RoboDK station: kr30 cnc 070419 2.rdk

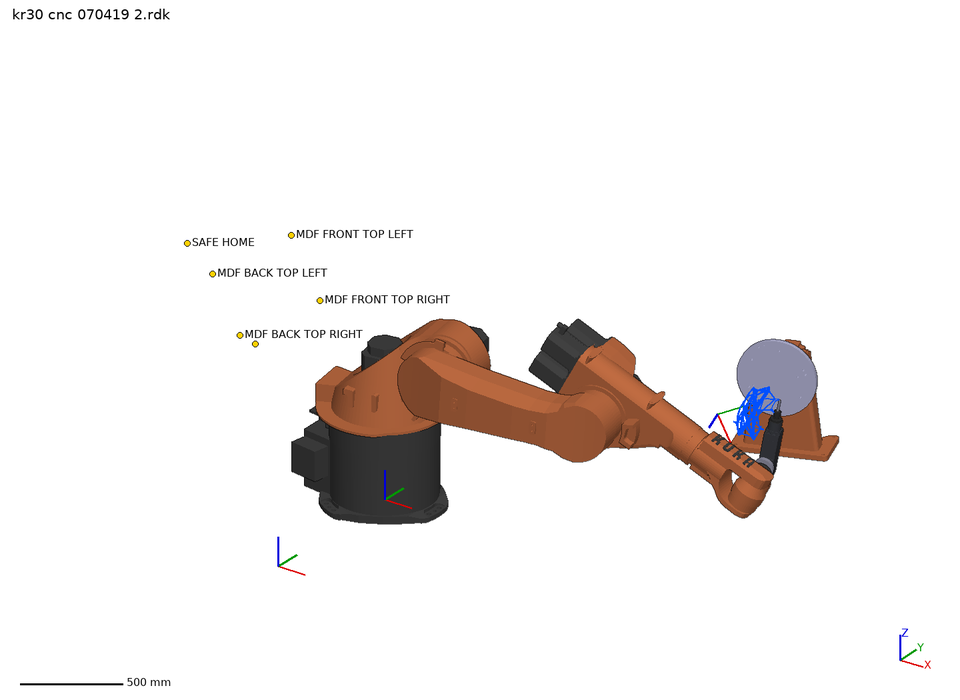
[picture v0: the station drawn from its stored meshes, robots at their saved joint values, targets as dots, program paths as lines]
Station kr30 cnc 070419 2. Poses are relative to the parent item; angles as X-Y-Z fixed-axis rotations.
  - frame GIGASHEEN 7th Axis Base at (0, 1100, 0) mm
    - robot KUKA KP1 MD250: 1 axes, payload 250 kg
        modified DH rows (alpha deg, a mm, theta deg, d mm): 0, 0, 0, 0
        base shift (1750, 1710, 820) mm, rotated rx 0 ry 90 rz -70 deg
        joint limits [-3600] to [3600]; home [0]; saved at [-335.665]
      - frame Reference Rhino at (0, -250, 250) mm
        - object RhinoPart at (0, 0, 0) mm
  - frame GIGASHEEN Base at (0, 2000, 0) mm
    - robot GIGASHEEN (model KUKA KR 30 HA): 6 axes, payload 30 kg, reach 2033 mm, repeatability 0.05 mm, weight 665 kg
        modified DH rows (alpha deg, a mm, theta deg, d mm): 0, 0, 0, 815; -90, 350, 0, 0; 0, 850, -90, 0; -90, 145, 0, 820; 90, 0, 0, 0; -90, 0, 180, 170
        joint limits [-185, -135, -120, -350, -119, -350] to [185, 35, 158, 350, 119, 350]; home [0, -90, 90, 0, 0, 0]; saved at [-7.883, 4.087, 23.625, 95.701, -100.709, 108.247]
      - tool 1/2" End Mill TCP, TCP at (337.71, -2.2, 160.57) mm, rotated rx 0 ry 90 rz 0 deg, size 415.8 x 102 x 153.6 mm
    - target MDF BACK TOP LEFT (joint target) at (-335.18, -974.02, 1512.92) mm, rotated rx 85.17 ry 71.84 rz 47.05 deg; joints [27.716, -45.008, 102.25, 116.233, 75.695, -151.59, -681.46] of GIGASHEEN
    - target MDF FRONT TOP LEFT (joint target) at (-87.97, -665.25, 1668.52) mm, rotated rx 85.17 ry 71.84 rz 47.05 deg; joints [22.06, -21.631, 54.581, 104.768, 70.881, -126.376, -681.46] of GIGASHEEN
    - target MDF FRONT TOP RIGHT (joint target) at (4.03, -550.6, 1295.2) mm, rotated rx 85.17 ry 71.84 rz 47.05 deg; joints [10.053, -29.315, 70.245, 98.928, 81.917, -132.341, -681.46] of GIGASHEEN
    - target MDF BACK TOP RIGHT (joint target) at (-248.73, -867.72, 1165.36) mm, rotated rx 85.17 ry 71.84 rz 47.05 deg; joints [13.787, -50.344, 113.459, 104.66, 84.215, -154.683, -681.46] of GIGASHEEN
    - target MDF STOCK DEPTH (only use z axis value) (joint target) at (-166.67, -856.91, 1136.76) mm, rotated rx 85.17 ry 71.84 rz 47.05 deg; joints [11.502, -45.737, 110.222, 102.707, 85.519, -155.78, -681.46] of GIGASHEEN
    - target SAFE HOME (joint target) at (-1073.3, -134.71, 1136.76) mm, rotated rx 85.17 ry 71.84 rz 47.05 deg; joints [11.502, -69.45, 58.776, 88.861, 76.585, -79.989, -681.46] of GIGASHEEN
  - machining project RhinoPart Settings: rotZ(0) | rotX(0)*rotY(270) | rotz(0) | onStart | onPathStart | onApproach | onPoint | onRetract | onFinish | onPathFinish | M_RunCode(%1)
  - program RhinoPart (845 instructions, listed below)
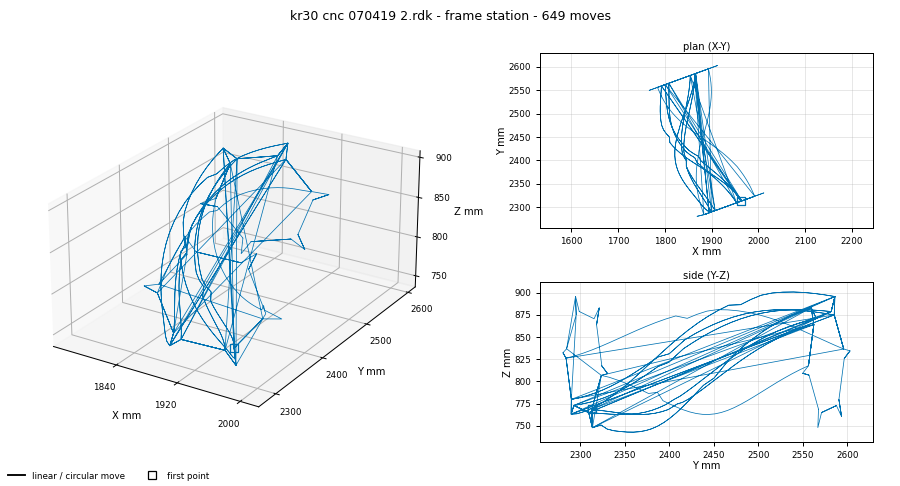
[picture p0: tool path of kr30 cnc 070419 2.rdk in frame station, 649 of 649 moves have a stored position in this frame; points joined in program order, loops and branches not executed]

--- program RhinoPart (robot GIGASHEEN) ---
  Set Ref.: Reference Rhino
  Set Tool: 1/2" End Mill TCP
  Show 1/2" End Mill TCP
  Set speed (1000.0 mm/s)
  MoveJ 1 to (58.93, 255.88, 290) mm, rotated rx 0 ry -90 rz -114.31 deg; joints [0.773, 4.57, 21.856, 99.582, -108.518, 97.992, -265.694]
  MoveL 2 to (58.93, 255.88, 290) mm, rotated rx 0 ry -90 rz -114.31 deg; joints [0.773, 4.57, 21.856, 99.582, -108.518, 97.992, -265.694]
  MoveL 3 to (58.93, 255.88, 290) mm, rotated rx 0 ry -90 rz -114.31 deg; joints [0.773, 4.57, 21.856, 99.582, -108.518, 97.992, -265.694]
  Set speed (60.0 mm/s)
  MoveL 4 to (37.11, 300.24, 290) mm, rotated rx 0 ry -90 rz -66.45 deg; joints [0.74, 5.545, 19.811, 99.211, -108.664, 96.873, -313.547]
  Set speed (1000.0 mm/s)
  MoveL 5 to (37.11, 300.24, 290) mm, rotated rx 0 ry -90 rz -66.45 deg; joints [0.74, 5.545, 19.811, 99.211, -108.664, 96.873, -313.547]
  Set speed (1000.0 mm/s)
  MoveL 6 to (-37.11, 208.63, 290) mm, rotated rx 0 ry -90 rz 108.11 deg; joints [0.809, 3.649, 23.804, 99.938, -108.376, 99.064, -488.107]
  MoveL 7 to (-37.11, 208.63, 290) mm, rotated rx 0 ry -90 rz 108.11 deg; joints [0.809, 3.649, 23.804, 99.938, -108.376, 99.064, -488.107]
  Set speed (60.0 mm/s)
  MoveL 8 to (-58.93, 252.99, 290) mm, rotated rx 0 ry -90 rz 57.1 deg; joints [0.775, 4.511, 21.98, 99.605, -108.509, 98.06, -437.096]
  Set speed (1000.0 mm/s)
  MoveL 9 to (-58.93, 252.99, 290) mm, rotated rx 0 ry -90 rz 57.1 deg; joints [0.775, 4.511, 21.98, 99.605, -108.509, 98.06, -437.096]
  Set speed (1000.0 mm/s)
  MoveL 10 to (21.11, 199.39, 290) mm, rotated rx 0 ry -90 rz 172.64 deg; joints [0.817, 3.477, 24.167, 100.005, -108.35, 99.264, -552.645]
  MoveL 11 to (21.11, 199.39, 290) mm, rotated rx 0 ry -90 rz 172.64 deg; joints [0.817, 3.477, 24.167, 100.005, -108.35, 99.264, -552.645]
  Set speed (60.0 mm/s)
  MoveL 12 to (34.26, 188.12, 288.36) mm, rotated rx 0 ry -90 rz 177.69 deg; joints [0.617, 10.244, 10.028, 97.427, -109.288, 91.536, -557.692]
  Set speed (1000.0 mm/s)
  MoveL 13 to (34.26, 188.12, 288.36) mm, rotated rx 0 ry -90 rz 177.69 deg; joints [0.617, 10.244, 10.028, 97.427, -109.288, 91.536, -557.692]
  Set speed (1000.0 mm/s)
  MoveL 14 to (21.11, 199.39, 290) mm, rotated rx 0 ry -90 rz 172.64 deg; joints [0.817, 3.477, 24.167, 100.005, -108.35, 99.264, -552.645]
  MoveL 15 to (21.11, 199.39, 290) mm, rotated rx 0 ry -90 rz 172.64 deg; joints [0.817, 3.477, 24.167, 100.005, -108.35, 99.264, -552.645]
  Set speed (60.0 mm/s)
  MoveL 16 to (-28.22, 202.67, 290) mm, rotated rx 0 ry -90 rz 119.2 deg; joints [0.814, 3.538, 24.039, 99.981, -108.359, 99.193, -499.196]
  Set speed (1000.0 mm/s)
  MoveL 17 to (-28.22, 202.67, 290) mm, rotated rx 0 ry -90 rz 119.2 deg; joints [0.814, 3.538, 24.039, 99.981, -108.359, 99.193, -499.196]
  Set speed (1000.0 mm/s)
  MoveL 18 to (-39.93, 191.53, 288.27) mm, rotated rx 0 ry -90 rz 114.31 deg; joints [0.614, 10.241, 10.028, 97.424, -109.285, 91.532, -494.314]
  MoveL 19 to (-39.93, 191.53, 288.27) mm, rotated rx 0 ry -90 rz 114.31 deg; joints [0.614, 10.241, 10.028, 97.424, -109.285, 91.532, -494.314]
  Set speed (60.0 mm/s)
  MoveL 20 to (-28.22, 202.67, 290) mm, rotated rx 0 ry -90 rz 119.2 deg; joints [0.814, 3.538, 24.039, 99.981, -108.359, 99.193, -499.196]
  Set speed (1000.0 mm/s)
  MoveL 21 to (-28.22, 202.67, 290) mm, rotated rx 0 ry -90 rz 119.2 deg; joints [0.814, 3.538, 24.039, 99.981, -108.359, 99.193, -499.196]
  Set speed (1000.0 mm/s)
  MoveL 22 to (-39.93, 191.53, 288.27) mm, rotated rx 0 ry -90 rz 114.31 deg; joints [0.614, 10.241, 10.028, 97.424, -109.285, 91.532, -494.314]
  MoveL 23 to (-39.93, 191.53, 288.27) mm, rotated rx 0 ry -90 rz 114.31 deg; joints [0.614, 10.241, 10.028, 97.424, -109.285, 91.532, -494.314]
  Set speed (60.0 mm/s)
  MoveL 24 to (-37.11, 208.63, 290) mm, rotated rx 0 ry -90 rz 108.11 deg; joints [0.809, 17.282, -3.748, 95.083, -110.206, 84.441, -488.107]
  Set speed (1000.0 mm/s)
  MoveL 25 to (-37.11, 208.63, 290) mm, rotated rx 0 ry -90 rz 108.11 deg; joints [0.809, 17.282, -3.748, 95.083, -110.206, 84.441, -488.107]
  Set speed (1000.0 mm/s)
  MoveL 26 to (-78.63, 259.66, 290) mm, rotated rx 0 ry -90 rz 42.99 deg; joints [1.123, 22.793, -16.516, 92.419, -110.99, 66.725, -432.994]
  MoveL 27 to (-78.63, 259.66, 290) mm, rotated rx 0 ry -90 rz 42.99 deg; joints [1.123, 22.793, -16.516, 92.419, -110.99, 66.725, -432.994]
  Set speed (60.0 mm/s)
  MoveL 28 to (-58.93, 252.99, 290) mm, rotated rx 0 ry -90 rz 57.1 deg; joints [0.775, 16.34, -1.924, 95.395, -110.092, 85.372, -437.096]
  Set speed (1000.0 mm/s)
  MoveL 29 to (-58.93, 252.99, 290) mm, rotated rx 0 ry -90 rz 57.1 deg; joints [0.775, 16.34, -1.924, 95.395, -110.092, 85.372, -437.096]
  Set speed (1000.0 mm/s)
  MoveL 30 to (-78.63, 259.66, 290) mm, rotated rx 0 ry -90 rz 42.99 deg; joints [1.123, 22.793, -16.516, 92.419, -110.99, 66.725, -432.994]
  MoveL 31 to (-78.63, 259.66, 290) mm, rotated rx 0 ry -90 rz 42.99 deg; joints [1.123, 22.793, -16.516, 92.419, -110.99, 66.725, -432.994]
  Set speed (60.0 mm/s)
  MoveL 32 to (-58.22, 263.67, 290) mm, rotated rx 0 ry -90 rz 46.79 deg; joints [0.767, 16.101, -1.46, 95.475, -110.063, 85.611, -426.787]
  Set speed (1000.0 mm/s)
  MoveL 33 to (-58.22, 263.67, 290) mm, rotated rx 0 ry -90 rz 46.79 deg; joints [0.767, 16.101, -1.46, 95.475, -110.063, 85.611, -426.787]
  Set speed (1000.0 mm/s)
  MoveL 34 to (-30.72, 304.75, 290) mm, rotated rx 0 ry -90 rz -0.71 deg; joints [0.737, 15.112, 0.47, 95.807, -109.942, 86.604, -379.294]
  MoveL 35 to (-30.72, 304.75, 290) mm, rotated rx 0 ry -90 rz -0.71 deg; joints [0.737, 15.112, 0.47, 95.807, -109.942, 86.604, -379.294]
  Set speed (60.0 mm/s)
  MoveL 36 to (-58.22, 263.67, 290) mm, rotated rx 0 ry -90 rz 46.79 deg; joints [0.767, 16.101, -1.46, 95.475, -110.063, 85.611, -426.787]
  Set speed (1000.0 mm/s)
  MoveL 37 to (-58.22, 263.67, 290) mm, rotated rx 0 ry -90 rz 46.79 deg; joints [0.767, 16.101, -1.46, 95.475, -110.063, 85.611, -426.787]
  Set speed (1000.0 mm/s)
  MoveL 38 to (-30.72, 304.75, 290) mm, rotated rx 0 ry -90 rz -0.71 deg; joints [0.737, 15.112, 0.47, 95.807, -109.942, 86.604, -379.294]
  MoveL 39 to (-30.72, 304.75, 290) mm, rotated rx 0 ry -90 rz -0.71 deg; joints [0.737, 15.112, 0.47, 95.807, -109.942, 86.604, -379.294]
  Set speed (60.0 mm/s)
  MoveL 40 to (-34.79, 325.15, 290) mm, rotated rx 0 ry -90 rz -15.16 deg; joints [1.086, 22.283, -15.568, 92.582, -110.934, 67.192, -374.84]
  Set speed (1000.0 mm/s)
  MoveL 41 to (-34.79, 325.15, 290) mm, rotated rx 0 ry -90 rz -15.16 deg; joints [1.086, 22.283, -15.568, 92.582, -110.934, 67.192, -374.84]
  Set speed (1000.0 mm/s)
  MoveL 42 to (-21.11, 309.47, 290) mm, rotated rx 0 ry -90 rz -10.46 deg; joints [0.734, 14.989, 0.711, 95.849, -109.927, 86.728, -369.544]
  MoveL 43 to (-21.11, 309.47, 290) mm, rotated rx 0 ry -90 rz -10.46 deg; joints [0.734, 14.989, 0.711, 95.849, -109.927, 86.728, -369.544]
  Set speed (60.0 mm/s)
  MoveL 44 to (-34.79, 325.15, 290) mm, rotated rx 0 ry -90 rz -15.16 deg; joints [1.086, 22.283, -15.568, 92.582, -110.934, 67.192, -374.84]
  Set speed (1000.0 mm/s)
  MoveL 45 to (-34.79, 325.15, 290) mm, rotated rx 0 ry -90 rz -15.16 deg; joints [1.086, 22.283, -15.568, 92.582, -110.934, 67.192, -374.84]
  Set speed (1000.0 mm/s)
  MoveL 46 to (-21.11, 309.47, 290) mm, rotated rx 0 ry -90 rz -10.46 deg; joints [0.734, 14.989, 0.711, 95.849, -109.927, 86.728, -369.544]
  MoveL 47 to (-21.11, 309.47, 290) mm, rotated rx 0 ry -90 rz -10.46 deg; joints [0.734, 14.989, 0.711, 95.849, -109.927, 86.728, -369.544]
  Set speed (60.0 mm/s)
  MoveL 48 to (28.22, 306.19, 290) mm, rotated rx 0 ry -90 rz -56.66 deg; joints [0.736, 15.075, 0.543, 95.82, -109.937, 86.642, -323.337]
  Set speed (1000.0 mm/s)
  MoveL 49 to (28.22, 306.19, 290) mm, rotated rx 0 ry -90 rz -56.66 deg; joints [0.736, 15.075, 0.543, 95.82, -109.937, 86.642, -323.337]
  Set speed (1000.0 mm/s)
  MoveL 50 to (43.85, 319.91, 290) mm, rotated rx 0 ry -90 rz -72.09 deg; joints [1.088, 22.324, -15.643, 92.569, -110.939, 67.155, -317.907]
  MoveL 51 to (43.85, 319.91, 290) mm, rotated rx 0 ry -90 rz -72.09 deg; joints [1.088, 22.324, -15.643, 92.569, -110.939, 67.155, -317.907]
  Set speed (60.0 mm/s)
  MoveL 52 to (28.22, 306.19, 290) mm, rotated rx 0 ry -90 rz -56.66 deg; joints [0.736, 15.075, 0.543, 95.82, -109.937, 86.642, -323.337]
  Set speed (1000.0 mm/s)
  MoveL 53 to (28.22, 306.19, 290) mm, rotated rx 0 ry -90 rz -56.66 deg; joints [0.736, 15.075, 0.543, 95.82, -109.937, 86.642, -323.337]
  Set speed (1000.0 mm/s)
  MoveL 54 to (43.85, 319.91, 290) mm, rotated rx 0 ry -90 rz -72.09 deg; joints [1.088, 22.324, -15.643, 92.569, -110.939, 67.155, -317.907]
  MoveL 55 to (43.85, 319.91, 290) mm, rotated rx 0 ry -90 rz -72.09 deg; joints [1.088, 22.324, -15.643, 92.569, -110.939, 67.155, -317.907]
  Set speed (60.0 mm/s)
  MoveL 56 to (37.11, 300.24, 290) mm, rotated rx 0 ry -90 rz -66.45 deg; joints [0.74, 15.227, 0.244, 95.768, -109.956, 86.487, -313.547]
  Set speed (1000.0 mm/s)
  MoveL 57 to (37.11, 300.24, 290) mm, rotated rx 0 ry -90 rz -66.45 deg; joints [0.74, 15.227, 0.244, 95.768, -109.956, 86.487, -313.547]
  Set speed (1000.0 mm/s)
  MoveL 58 to (78.63, 249.2, 290) mm, rotated rx 0 ry -90 rz -130.58 deg; joints [1.129, 22.875, -16.669, 92.392, -110.999, 66.65, -259.419]
  MoveL 59 to (78.63, 249.2, 290) mm, rotated rx 0 ry -90 rz -130.58 deg; joints [1.129, 22.875, -16.669, 92.392, -110.999, 66.65, -259.419]
  Set speed (60.0 mm/s)
  MoveL 60 to (58.93, 255.88, 290) mm, rotated rx 0 ry -90 rz -114.31 deg; joints [0.773, 16.276, -1.8, 95.417, -110.084, 85.436, -265.694]
  Set speed (1000.0 mm/s)
  MoveL 61 to (58.93, 255.88, 290) mm, rotated rx 0 ry -90 rz -114.31 deg; joints [0.773, 16.276, -1.8, 95.417, -110.084, 85.436, -265.694]
  Set speed (1000.0 mm/s)
  MoveL 62 to (78.63, 249.2, 290) mm, rotated rx 0 ry -90 rz -130.58 deg; joints [1.129, 22.875, -16.669, 92.392, -110.999, 66.65, -259.419]
  MoveL 63 to (78.63, 249.2, 290) mm, rotated rx 0 ry -90 rz -130.58 deg; joints [1.129, 22.875, -16.669, 92.392, -110.999, 66.65, -259.419]
  Set speed (60.0 mm/s)
  MoveL 64 to (58.22, 245.2, 290) mm, rotated rx 0 ry -90 rz -124.72 deg; joints [0.781, 16.511, -2.256, 95.338, -110.113, 85.202, -255.284]
  Set speed (1000.0 mm/s)
  MoveL 65 to (58.22, 245.2, 290) mm, rotated rx 0 ry -90 rz -124.72 deg; joints [0.781, 16.511, -2.256, 95.338, -110.113, 85.202, -255.284]
  Set speed (1000.0 mm/s)
  MoveL 66 to (30.72, 204.12, 290) mm, rotated rx 0 ry -90 rz -176.2 deg; joints [0.813, 17.375, -3.926, 95.052, -110.217, 84.35, -203.801]
  MoveL 67 to (30.72, 204.12, 290) mm, rotated rx 0 ry -90 rz -176.2 deg; joints [0.813, 17.375, -3.926, 95.052, -110.217, 84.35, -203.801]
  Set speed (60.0 mm/s)
  MoveL 68 to (58.22, 245.2, 290) mm, rotated rx 0 ry -90 rz -124.72 deg; joints [0.781, 16.511, -2.256, 95.338, -110.113, 85.202, -255.284]
  Set speed (1000.0 mm/s)
  MoveL 69 to (58.22, 245.2, 290) mm, rotated rx 0 ry -90 rz -124.72 deg; joints [0.781, 16.511, -2.256, 95.338, -110.113, 85.202, -255.284]
  Set speed (1000.0 mm/s)
  MoveL 70 to (30.72, 204.12, 290) mm, rotated rx 0 ry -90 rz -176.2 deg; joints [0.813, 17.375, -3.926, 95.052, -110.217, 84.35, -203.801]
  MoveL 71 to (30.72, 204.12, 290) mm, rotated rx 0 ry -90 rz -176.2 deg; joints [0.813, 17.375, -3.926, 95.052, -110.217, 84.35, -203.801]
  Set speed (60.0 mm/s)
  MoveL 72 to (34.26, 188.12, 288.36) mm, rotated rx 0 ry -90 rz 177.69 deg; joints [0.617, 10.244, 10.028, 97.427, -109.288, 91.536, -197.692]
  Set speed (1000.0 mm/s)
  MoveL 73 to (34.26, 188.12, 288.36) mm, rotated rx 0 ry -90 rz 177.69 deg; joints [0.617, 10.244, 10.028, 97.427, -109.288, 91.536, -197.692]
  Set speed (1000.0 mm/s)
  MoveL 74 to (-37.62, 299.82, 0) mm, rotated rx 0 ry -90 rz 17.06 deg; joints [-7.759, 0.223, 31.945, 96.589, -100.339, 112.764, -27.061]
  MoveL 75 to (-37.62, 299.82, 0) mm, rotated rx 0 ry -90 rz 17.06 deg; joints [-7.759, 0.223, 31.945, 96.589, -100.339, 112.764, -27.061]
  Set speed (60.0 mm/s)
  MoveL 76 to (10.16, 312.5, 0) mm, rotated rx 0 ry -90 rz -29.23 deg; joints [-7.765, 0.357, 31.651, 96.557, -100.353, 112.603, 19.233]
  Set speed (1000.0 mm/s)
  MoveL 77 to (10.16, 312.5, 0) mm, rotated rx 0 ry -90 rz -29.23 deg; joints [-7.765, 0.357, 31.651, 96.557, -100.353, 112.603, 19.233]
  Set speed (1000.0 mm/s)
  MoveL 78 to (-37.62, 299.82, 0) mm, rotated rx 0 ry -90 rz 17.06 deg; joints [-7.759, 0.223, 31.945, 96.589, -100.339, 112.764, -27.061]
  MoveL 79 to (-37.62, 299.82, 0) mm, rotated rx 0 ry -90 rz 17.06 deg; joints [-7.759, 0.223, 31.945, 96.589, -100.339, 112.764, -27.061]
  Set speed (60.0 mm/s)
  MoveL 80 to (-55.59, 310.29, 0) mm, rotated rx 0 ry -90 rz 22.68 deg; joints [-7.877, 3.824, 24.184, 95.76, -100.685, 108.547, -32.681]
  Set speed (1000.0 mm/s)
  MoveL 81 to (-55.59, 310.29, 0) mm, rotated rx 0 ry -90 rz 22.68 deg; joints [-7.877, 3.824, 24.184, 95.76, -100.685, 108.547, -32.681]
  Set speed (1000.0 mm/s)
  MoveL 82 to (-45.21, 292.27, 0) mm, rotated rx 0 ry -90 rz 26.93 deg; joints [-7.756, 0.143, 32.12, 96.608, -100.331, 112.861, -36.927]
  MoveL 83 to (-45.21, 292.27, 0) mm, rotated rx 0 ry -90 rz 26.93 deg; joints [-7.756, 0.143, 32.12, 96.608, -100.331, 112.861, -36.927]
  Set speed (60.0 mm/s)
  MoveL 84 to (-55.59, 310.29, 0) mm, rotated rx 0 ry -90 rz 22.68 deg; joints [-7.877, 3.824, 24.184, 95.76, -100.685, 108.547, -32.681]
  Set speed (1000.0 mm/s)
  MoveL 85 to (-55.59, 310.29, 0) mm, rotated rx 0 ry -90 rz 22.68 deg; joints [-7.877, 3.824, 24.184, 95.76, -100.685, 108.547, -32.681]
  Set speed (1000.0 mm/s)
  MoveL 86 to (-45.21, 292.27, 0) mm, rotated rx 0 ry -90 rz 26.93 deg; joints [-7.756, 0.143, 32.12, 96.608, -100.331, 112.861, -36.927]
  MoveL 87 to (-45.21, 292.27, 0) mm, rotated rx 0 ry -90 rz 26.93 deg; joints [-7.756, 0.143, 32.12, 96.608, -100.331, 112.861, -36.927]
  Set speed (60.0 mm/s)
  MoveL 88 to (-58.12, 244.54, 0) mm, rotated rx 0 ry -90 rz 75.36 deg; joints [-7.735, -0.364, 33.232, 96.729, -100.279, 113.474, -85.364]
  Set speed (1000.0 mm/s)
  MoveL 89 to (-58.12, 244.54, 0) mm, rotated rx 0 ry -90 rz 75.36 deg; joints [-7.735, -0.364, 33.232, 96.729, -100.279, 113.474, -85.364]
  Set speed (1000.0 mm/s)
  MoveL 90 to (-76.17, 234.21, 0) mm, rotated rx 0 ry -90 rz 81.71 deg; joints [-7.852, 2.89, 26.175, 95.97, -100.599, 109.619, -91.709]
  MoveL 91 to (-76.17, 234.21, 0) mm, rotated rx 0 ry -90 rz 81.71 deg; joints [-7.852, 2.89, 26.175, 95.97, -100.599, 109.619, -91.709]
  Set speed (60.0 mm/s)
  MoveL 92 to (-58.12, 244.54, 0) mm, rotated rx 0 ry -90 rz 75.36 deg; joints [-7.735, -0.364, 33.232, 96.729, -100.279, 113.474, -85.364]
  Set speed (1000.0 mm/s)
  MoveL 93 to (-58.12, 244.54, 0) mm, rotated rx 0 ry -90 rz 75.36 deg; joints [-7.735, -0.364, 33.232, 96.729, -100.279, 113.474, -85.364]
  Set speed (1000.0 mm/s)
  MoveL 94 to (-76.17, 234.21, 0) mm, rotated rx 0 ry -90 rz 81.71 deg; joints [-7.852, 2.89, 26.175, 95.97, -100.599, 109.619, -91.709]
  MoveL 95 to (-76.17, 234.21, 0) mm, rotated rx 0 ry -90 rz 81.71 deg; joints [-7.852, 2.89, 26.175, 95.97, -100.599, 109.619, -91.709]
  Set speed (60.0 mm/s)
  MoveL 96 to (-55.37, 234.2, 0) mm, rotated rx 0 ry -90 rz 85.93 deg; joints [-7.73, -0.474, 33.474, 96.756, -100.267, 113.608, -95.929]
  Set speed (1000.0 mm/s)
  MoveL 97 to (-55.37, 234.2, 0) mm, rotated rx 0 ry -90 rz 85.93 deg; joints [-7.73, -0.474, 33.474, 96.756, -100.267, 113.608, -95.929]
  Set speed (1000.0 mm/s)
  MoveL 98 to (-20.49, 199.16, 0) mm, rotated rx 0 ry -90 rz 138.05 deg; joints [-7.713, -0.85, 34.304, 96.846, -100.227, 114.067, -148.047]
  MoveL 99 to (-20.49, 199.16, 0) mm, rotated rx 0 ry -90 rz 138.05 deg; joints [-7.713, -0.85, 34.304, 96.846, -100.227, 114.067, -148.047]
  Set speed (60.0 mm/s)
  MoveL 100 to (-55.37, 234.2, 0) mm, rotated rx 0 ry -90 rz 85.93 deg; joints [-7.73, -0.474, 33.474, 96.756, -100.267, 113.608, -95.929]
  Set speed (1000.0 mm/s)
  MoveL 101 to (-55.37, 234.2, 0) mm, rotated rx 0 ry -90 rz 85.93 deg; joints [-7.73, -0.474, 33.474, 96.756, -100.267, 113.608, -95.929]
  Set speed (1000.0 mm/s)
  MoveL 102 to (-20.49, 199.16, 0) mm, rotated rx 0 ry -90 rz 138.05 deg; joints [-7.713, -0.85, 34.304, 96.846, -100.227, 114.067, -148.047]
  MoveL 103 to (-20.49, 199.16, 0) mm, rotated rx 0 ry -90 rz 138.05 deg; joints [-7.713, -0.85, 34.304, 96.846, -100.227, 114.067, -148.047]
  Set speed (60.0 mm/s)
  MoveL 104 to (-20.57, 178.36, 0) mm, rotated rx 0 ry -90 rz 143.98 deg; joints [-7.832, 2.246, 27.555, 96.116, -100.539, 110.366, -153.977]
  Set speed (1000.0 mm/s)
  MoveL 105 to (-20.57, 178.36, 0) mm, rotated rx 0 ry -90 rz 143.98 deg; joints [-7.832, 2.246, 27.555, 96.116, -100.539, 110.366, -153.977]
  Set speed (1000.0 mm/s)
  MoveL 106 to (-10.16, 196.36, 0) mm, rotated rx 0 ry -90 rz 149.27 deg; joints [-7.711, -0.88, 34.37, 96.854, -100.224, 114.104, -159.273]
  MoveL 107 to (-10.16, 196.36, 0) mm, rotated rx 0 ry -90 rz 149.27 deg; joints [-7.711, -0.88, 34.37, 96.854, -100.224, 114.104, -159.273]
  Set speed (60.0 mm/s)
  MoveL 108 to (-20.57, 178.36, 0) mm, rotated rx 0 ry -90 rz 143.98 deg; joints [-7.832, 2.246, 27.555, 96.116, -100.539, 110.366, -153.977]
  Set speed (1000.0 mm/s)
  MoveL 109 to (-20.57, 178.36, 0) mm, rotated rx 0 ry -90 rz 143.98 deg; joints [-7.832, 2.246, 27.555, 96.116, -100.539, 110.366, -153.977]
  Set speed (1000.0 mm/s)
  MoveL 110 to (-10.16, 196.36, 0) mm, rotated rx 0 ry -90 rz 149.27 deg; joints [-7.711, -0.88, 34.37, 96.854, -100.224, 114.104, -159.273]
  MoveL 111 to (-10.16, 196.36, 0) mm, rotated rx 0 ry -90 rz 149.27 deg; joints [-7.711, -0.88, 34.37, 96.854, -100.224, 114.104, -159.273]
  Set speed (60.0 mm/s)
  MoveL 112 to (37.62, 209.05, 0) mm, rotated rx 0 ry -90 rz -157.43 deg; joints [-7.718, -0.743, 34.068, 96.821, -100.239, 113.937, -212.574]
  Set speed (1000.0 mm/s)
  MoveL 113 to (37.62, 209.05, 0) mm, rotated rx 0 ry -90 rz -157.43 deg; joints [-7.718, -0.743, 34.068, 96.821, -100.239, 113.937, -212.574]
  Set speed (1000.0 mm/s)
  MoveL 114 to (55.59, 198.58, 0) mm, rotated rx 0 ry -90 rz -152.77 deg; joints [-7.839, 2.476, 27.061, 96.064, -100.561, 110.098, -217.234]
  MoveL 115 to (55.59, 198.58, 0) mm, rotated rx 0 ry -90 rz -152.77 deg; joints [-7.839, 2.476, 27.061, 96.064, -100.561, 110.098, -217.234]
  Set speed (60.0 mm/s)
  MoveL 116 to (37.62, 209.05, 0) mm, rotated rx 0 ry -90 rz -157.43 deg; joints [-7.718, -0.743, 34.068, 96.821, -100.239, 113.937, -212.574]
  Set speed (1000.0 mm/s)
  MoveL 117 to (37.62, 209.05, 0) mm, rotated rx 0 ry -90 rz -157.43 deg; joints [-7.718, -0.743, 34.068, 96.821, -100.239, 113.937, -212.574]
  Set speed (1000.0 mm/s)
  MoveL 118 to (55.59, 198.58, 0) mm, rotated rx 0 ry -90 rz -152.77 deg; joints [-7.839, 2.476, 27.061, 96.064, -100.561, 110.098, -217.234]
  MoveL 119 to (55.59, 198.58, 0) mm, rotated rx 0 ry -90 rz -152.77 deg; joints [-7.839, 2.476, 27.061, 96.064, -100.561, 110.098, -217.234]
  Set speed (60.0 mm/s)
  MoveL 120 to (45.21, 216.6, 0) mm, rotated rx 0 ry -90 rz -146.46 deg; joints [-7.721, -0.662, 33.889, 96.801, -100.247, 113.838, -223.543]
  Set speed (1000.0 mm/s)
  MoveL 121 to (45.21, 216.6, 0) mm, rotated rx 0 ry -90 rz -146.46 deg; joints [-7.721, -0.662, 33.889, 96.801, -100.247, 113.838, -223.543]
  Set speed (1000.0 mm/s)
  MoveL 122 to (58.12, 264.32, 0) mm, rotated rx 0 ry -90 rz -96.15 deg; joints [-7.744, -0.154, 32.77, 96.679, -100.3, 113.219, -273.845]
  MoveL 123 to (58.12, 264.32, 0) mm, rotated rx 0 ry -90 rz -96.15 deg; joints [-7.744, -0.154, 32.77, 96.679, -100.3, 113.219, -273.845]
  Set speed (60.0 mm/s)
  MoveL 124 to (45.21, 216.6, 0) mm, rotated rx 0 ry -90 rz -146.46 deg; joints [-7.721, -0.662, 33.889, 96.801, -100.247, 113.838, -223.543]
  Set speed (1000.0 mm/s)
  MoveL 125 to (45.21, 216.6, 0) mm, rotated rx 0 ry -90 rz -146.46 deg; joints [-7.721, -0.662, 33.889, 96.801, -100.247, 113.838, -223.543]
  Set speed (1000.0 mm/s)
  MoveL 126 to (58.12, 264.32, 0) mm, rotated rx 0 ry -90 rz -96.15 deg; joints [-7.744, -0.154, 32.77, 96.679, -100.3, 113.219, -273.845]
  MoveL 127 to (58.12, 264.32, 0) mm, rotated rx 0 ry -90 rz -96.15 deg; joints [-7.744, -0.154, 32.77, 96.679, -100.3, 113.219, -273.845]
  Set speed (60.0 mm/s)
  MoveL 128 to (76.17, 274.65, 0) mm, rotated rx 0 ry -90 rz -92.07 deg; joints [-7.865, 3.376, 25.136, 95.86, -100.645, 109.058, -277.935]
  Set speed (1000.0 mm/s)
  MoveL 129 to (76.17, 274.65, 0) mm, rotated rx 0 ry -90 rz -92.07 deg; joints [-7.865, 3.376, 25.136, 95.86, -100.645, 109.058, -277.935]
  Set speed (1000.0 mm/s)
  MoveL 130 to (55.37, 274.67, 0) mm, rotated rx 0 ry -90 rz -85.99 deg; joints [-7.748, -0.044, 32.529, 96.652, -100.312, 113.086, -284.014]
  MoveL 131 to (55.37, 274.67, 0) mm, rotated rx 0 ry -90 rz -85.99 deg; joints [-7.748, -0.044, 32.529, 96.652, -100.312, 113.086, -284.014]
  Set speed (60.0 mm/s)
  MoveL 132 to (76.17, 274.65, 0) mm, rotated rx 0 ry -90 rz -92.07 deg; joints [-7.865, 3.376, 25.136, 95.86, -100.645, 109.058, -277.935]
  Set speed (1000.0 mm/s)
  MoveL 133 to (76.17, 274.65, 0) mm, rotated rx 0 ry -90 rz -92.07 deg; joints [-7.865, 3.376, 25.136, 95.86, -100.645, 109.058, -277.935]
  Set speed (1000.0 mm/s)
  MoveL 134 to (55.37, 274.67, 0) mm, rotated rx 0 ry -90 rz -85.99 deg; joints [-7.748, -0.044, 32.529, 96.652, -100.312, 113.086, -284.014]
  MoveL 135 to (55.37, 274.67, 0) mm, rotated rx 0 ry -90 rz -85.99 deg; joints [-7.748, -0.044, 32.529, 96.652, -100.312, 113.086, -284.014]
  Set speed (60.0 mm/s)
  MoveL 136 to (20.49, 309.71, 0) mm, rotated rx 0 ry -90 rz -38.94 deg; joints [-7.763, 0.327, 31.716, 96.564, -100.35, 112.638, -331.057]
  Set speed (1000.0 mm/s)
  MoveL 137 to (20.49, 309.71, 0) mm, rotated rx 0 ry -90 rz -38.94 deg; joints [-7.763, 0.327, 31.716, 96.564, -100.35, 112.638, -331.057]
  Set speed (1000.0 mm/s)
  MoveL 138 to (20.57, 330.51, 0) mm, rotated rx 0 ry -90 rz -34.34 deg; joints [-7.883, 4.087, 23.625, 95.701, -100.709, 108.247, -335.665]
  MoveL 139 to (20.57, 330.51, 0) mm, rotated rx 0 ry -90 rz -34.34 deg; joints [-7.883, 4.087, 23.625, 95.701, -100.709, 108.247, -335.665]
  Set speed (60.0 mm/s)
  MoveL 140 to (20.49, 309.71, 0) mm, rotated rx 0 ry -90 rz -38.94 deg; joints [-7.763, 0.327, 31.716, 96.564, -100.35, 112.638, -331.057]
  Set speed (1000.0 mm/s)
  MoveL 141 to (20.49, 309.71, 0) mm, rotated rx 0 ry -90 rz -38.94 deg; joints [-7.763, 0.327, 31.716, 96.564, -100.35, 112.638, -331.057]
  Set speed (1000.0 mm/s)
  MoveL 142 to (20.57, 330.51, 0) mm, rotated rx 0 ry -90 rz -34.34 deg; joints [-7.883, 4.087, 23.625, 95.701, -100.709, 108.247, -335.665]
  MoveL 143 to (20.57, 330.51, 0) mm, rotated rx 0 ry -90 rz -34.34 deg; joints [-7.883, 4.087, 23.625, 95.701, -100.709, 108.247, -335.665]
  Set speed (60.0 mm/s)
  MoveL 144 to (10.16, 312.5, 0) mm, rotated rx 0 ry -90 rz -29.23 deg; joints [-7.765, 0.357, 31.651, 96.557, -100.353, 112.603, -340.767]
  Set speed (1000.0 mm/s)
  MoveL 145 to (10.16, 312.5, 0) mm, rotated rx 0 ry -90 rz -29.23 deg; joints [-7.765, 0.357, 31.651, 96.557, -100.353, 112.603, -340.767]
  Set speed (1000.0 mm/s)
  MoveL 146 to (-37.62, 299.82, 0) mm, rotated rx 0 ry -90 rz 17.06 deg; joints [-7.759, 0.223, 31.945, 96.589, -100.339, 112.764, -387.061]
  MoveL 147 to (-37.62, 299.82, 0) mm, rotated rx 0 ry -90 rz 17.06 deg; joints [-7.759, 0.223, 31.945, 96.589, -100.339, 112.764, -387.061]
  Set speed (60.0 mm/s)
  MoveL 148 to (-40.85, 296.93, 10) mm, rotated rx 0 ry -90 rz 21.04 deg; joints [-7.474, 0.556, 31.247, 96.678, -100.621, 112.424, -391.039]
  MoveL 149 to (-44.15, 293.5, 20) mm, rotated rx 0 ry -90 rz 25.42 deg; joints [-7.19, 0.904, 30.521, 96.761, -100.906, 112.071, -395.425]
  MoveL 150 to (-47.39, 289.5, 30) mm, rotated rx 0 ry -90 rz 30.19 deg; joints [-6.905, 1.267, 29.765, 96.838, -101.194, 111.702, -400.19]
  MoveL 151 to (-50.45, 284.92, 40) mm, rotated rx 0 ry -90 rz 35.31 deg; joints [-6.621, 1.646, 28.975, 96.908, -101.486, 111.316, -405.308]
  MoveL 152 to (-53.21, 279.8, 50) mm, rotated rx 0 ry -90 rz 40.75 deg; joints [-6.337, 2.045, 28.146, 96.97, -101.781, 110.911, -410.751]
  MoveL 153 to (-55.55, 274.16, 60) mm, rotated rx 0 ry -90 rz 46.49 deg; joints [-6.054, 2.466, 27.273, 97.023, -102.079, 110.484, -416.493]
  MoveL 154 to (-57.35, 268.08, 70) mm, rotated rx 0 ry -90 rz 52.51 deg; joints [-5.771, 2.914, 26.347, 97.066, -102.383, 110.029, -422.507]
  MoveL 155 to (-58.51, 261.62, 80) mm, rotated rx 0 ry -90 rz 58.76 deg; joints [-5.488, 3.395, 25.355, 97.097, -102.691, 109.54, -428.765]
  MoveL 156 to (-58.95, 254.91, 90) mm, rotated rx 0 ry -90 rz 65.24 deg; joints [-5.205, 3.916, 24.28, 97.113, -103.006, 109.008, -435.24]
  MoveL 157 to (-58.6, 248.05, 100) mm, rotated rx 0 ry -90 rz 71.9 deg; joints [-4.923, 4.491, 23.097, 97.111, -103.329, 108.42, -441.902]
  MoveL 158 to (-57.44, 241.19, 110) mm, rotated rx 0 ry -90 rz 78.72 deg; joints [-4.642, 5.137, 21.769, 97.085, -103.661, 107.755, -448.721]
  MoveL 159 to (-55.46, 234.45, 120) mm, rotated rx 0 ry -90 rz 85.66 deg; joints [-4.361, 5.887, 20.23, 97.025, -104.007, 106.981, -455.664]
  MoveL 160 to (-52.68, 227.97, 130) mm, rotated rx 0 ry -90 rz 92.7 deg; joints [-4.081, 6.802, 18.358, 96.914, -104.374, 106.033, -462.696]
  MoveL 161 to (-49.15, 221.88, 140) mm, rotated rx 0 ry -90 rz 99.78 deg; joints [-3.802, 8.043, 15.826, 96.704, -104.779, 104.739, -469.78]
  MoveL 162 to (-44.74, 216.34, 149.94) mm, rotated rx 0 ry -90 rz 106.88 deg; joints [-3.524, 10.899, 10.028, 96.03, -105.361, 101.741, -476.877]
  MoveL 163 to (-37.8, 212.27, 159.24) mm, rotated rx 0 ry -90 rz 113.94 deg; joints [-3.247, 10.885, 10.028, 96.133, -105.62, 101.755, -483.944]
  MoveL 164 to (-30.59, 209.42, 168.5) mm, rotated rx 0 ry -90 rz 120.94 deg; joints [-2.971, 10.871, 10.028, 96.235, -105.878, 101.769, -490.939]
  MoveL 165 to (-29.38, 203.32, 180) mm, rotated rx 0 ry -90 rz 117.81 deg; joints [-2.2, 24.317, -17.489, 92.186, -107.67, 77.167, -497.814]
  MoveL 166 to (-23.62, 200.42, 190) mm, rotated rx 0 ry -90 rz 124.52 deg; joints [-1.919, 23.894, -16.67, 92.351, -107.933, 77.595, -504.525]
  MoveL 167 to (-17.8, 198.23, 200) mm, rotated rx 0 ry -90 rz 131.02 deg; joints [-1.64, 23.444, -15.796, 92.529, -108.191, 78.053, -511.023]
  MoveL 168 to (-12.04, 196.73, 210) mm, rotated rx 0 ry -90 rz 137.26 deg; joints [-1.362, 22.963, -14.862, 92.721, -108.445, 78.543, -517.262]
  MoveL 169 to (-6.46, 195.84, 220) mm, rotated rx 0 ry -90 rz 143.2 deg; joints [-1.085, 22.449, -13.862, 92.929, -108.695, 79.069, -523.197]
  MoveL 170 to (-1.16, 195.49, 230) mm, rotated rx 0 ry -90 rz 148.78 deg; joints [-0.81, 21.898, -12.791, 93.153, -108.939, 79.633, -528.782]
  MoveL 171 to (3.78, 195.6, 240) mm, rotated rx 0 ry -90 rz 153.97 deg; joints [-0.536, 21.307, -11.64, 93.396, -109.176, 80.242, -533.974]
  MoveL 172 to (8.28, 196.07, 250) mm, rotated rx 0 ry -90 rz 158.73 deg; joints [-0.263, 20.671, -10.398, 93.661, -109.407, 80.9, -538.733]
  MoveL 173 to (12.3, 196.78, 260) mm, rotated rx 0 ry -90 rz 163.02 deg; joints [0.008, 19.983, -9.05, 93.95, -109.63, 81.616, -543.017]
  MoveL 174 to (15.8, 197.64, 270) mm, rotated rx 0 ry -90 rz 166.79 deg; joints [0.279, 19.231, -7.578, 94.268, -109.843, 82.401, -546.788]
  MoveL 175 to (18.74, 198.54, 280) mm, rotated rx 0 ry -90 rz 170.01 deg; joints [0.548, 18.402, -5.948, 94.622, -110.044, 83.272, -550.01]
  MoveL 176 to (21.11, 199.39, 290) mm, rotated rx 0 ry -90 rz 172.64 deg; joints [0.817, 17.471, -4.111, 95.02, -110.229, 84.256, -552.645]
  Set speed (1000.0 mm/s)
  MoveL 177 to (21.11, 199.39, 290) mm, rotated rx 0 ry -90 rz 172.64 deg; joints [0.817, 17.471, -4.111, 95.02, -110.229, 84.256, -552.645]
  Set speed (1000.0 mm/s)
  MoveL 178 to (10.16, 312.5, 0) mm, rotated rx 0 ry -90 rz -29.23 deg; joints [-7.765, 21.755, -11.595, 92.191, -102.041, 90.391, -700.767]
  MoveL 179 to (10.16, 312.5, 0) mm, rotated rx 0 ry -90 rz -29.23 deg; joints [-7.765, 21.755, -11.595, 92.191, -102.041, 90.391, -700.767]
  Set speed (60.0 mm/s)
  MoveL 180 to (-37.62, 299.82, 0) mm, rotated rx 0 ry -90 rz 17.06 deg; joints [-7.759, 21.912, -11.889, 92.162, -102.051, 90.251, -747.061]
  Set speed (1000.0 mm/s)
  MoveL 181 to (-37.62, 299.82, 0) mm, rotated rx 0 ry -90 rz 17.06 deg; joints [-7.759, 21.912, -11.889, 92.162, -102.051, 90.251, -747.061]
  Set speed (1000.0 mm/s)
  MoveL 182 to (-28.22, 202.67, 290) mm, rotated rx 0 ry -90 rz 119.2 deg; joints [0.814, 17.404, -3.983, 95.042, -110.221, 84.321, -859.196]
  MoveL 183 to (-28.22, 202.67, 290) mm, rotated rx 0 ry -90 rz 119.2 deg; joints [0.814, 17.404, -3.983, 95.042, -110.221, 84.321, -859.196]
  Set speed (60.0 mm/s)
  MoveL 184 to (21.11, 199.39, 290) mm, rotated rx 0 ry -90 rz 172.64 deg; joints [0.817, 17.471, -4.111, 95.02, -110.229, 84.256, -912.645]
  Set speed (1000.0 mm/s)
  MoveL 185 to (21.11, 199.39, 290) mm, rotated rx 0 ry -90 rz 172.64 deg; joints [0.817, 17.471, -4.111, 95.02, -110.229, 84.256, -912.645]
  Set speed (1000.0 mm/s)
  MoveL 186 to (-28.22, 202.67, 290) mm, rotated rx 0 ry -90 rz 119.2 deg; joints [0.814, 17.404, -3.983, 95.042, -110.221, 84.321, -859.196]
  MoveL 187 to (-28.22, 202.67, 290) mm, rotated rx 0 ry -90 rz 119.2 deg; joints [0.814, 17.404, -3.983, 95.042, -110.221, 84.321, -859.196]
  Set speed (60.0 mm/s)
  MoveL 188 to (-30.4, 203.93, 280) mm, rotated rx 0 ry -90 rz 116.58 deg; joints [0.544, 18.305, -5.761, 94.653, -110.032, 83.366, -856.579]
  MoveL 189 to (-33, 205.58, 270) mm, rotated rx 0 ry -90 rz 113.39 deg; joints [0.272, 19.099, -7.326, 94.31, -109.828, 82.527, -853.391]
  MoveL 190 to (-35.92, 207.69, 260) mm, rotated rx 0 ry -90 rz 109.67 deg; joints [0, 19.814, -8.731, 94.002, -109.611, 81.775, -849.674]
  MoveL 191 to (-39.07, 210.28, 250) mm, rotated rx 0 ry -90 rz 105.47 deg; joints [-0.274, 20.465, -10.008, 93.723, -109.385, 81.093, -845.473]
  MoveL 192 to (-42.34, 213.41, 240) mm, rotated rx 0 ry -90 rz 100.83 deg; joints [-0.55, 21.062, -11.179, 93.469, -109.15, 80.469, -840.831]
  MoveL 193 to (-45.62, 217.1, 230) mm, rotated rx 0 ry -90 rz 95.79 deg; joints [-0.826, 21.615, -12.26, 93.235, -108.909, 79.894, -835.794]
  MoveL 194 to (-48.8, 221.36, 220) mm, rotated rx 0 ry -90 rz 90.41 deg; joints [-1.104, 22.128, -13.263, 93.02, -108.662, 79.361, -830.406]
  MoveL 195 to (-51.74, 226.19, 210) mm, rotated rx 0 ry -90 rz 84.71 deg; joints [-1.383, 22.607, -14.198, 92.82, -108.409, 78.866, -824.713]
  MoveL 196 to (-54.33, 231.55, 200) mm, rotated rx 0 ry -90 rz 78.76 deg; joints [-1.664, 23.055, -15.074, 92.635, -108.153, 78.402, -818.758]
  MoveL 197 to (-56.44, 237.4, 190) mm, rotated rx 0 ry -90 rz 72.59 deg; joints [-1.945, 23.477, -15.897, 92.462, -107.892, 77.968, -812.587]
  MoveL 198 to (-57.96, 243.66, 180) mm, rotated rx 0 ry -90 rz 66.24 deg; joints [-2.227, 23.876, -16.675, 92.301, -107.628, 77.558, -806.24]
  MoveL 199 to (-58.8, 250.25, 170) mm, rotated rx 0 ry -90 rz 59.76 deg; joints [-2.511, 24.254, -17.412, 92.15, -107.361, 77.171, -799.76]
  MoveL 200 to (-53.97, 254.41, 158.36) mm, rotated rx 0 ry -90 rz 63.18 deg; joints [-3.275, 10.844, 10.028, 96.111, -105.598, 101.709, -793.183]
  MoveL 201 to (-55.44, 262.01, 149.03) mm, rotated rx 0 ry -90 rz 56.55 deg; joints [-3.553, 10.856, 10.028, 96.007, -105.339, 101.694, -786.549]
  MoveL 202 to (-55.81, 270, 139.68) mm, rotated rx 0 ry -90 rz 49.89 deg; joints [-3.831, 10.868, 10.028, 95.904, -105.079, 101.678, -779.89]
  MoveL 203 to (-54.3, 277.38, 130) mm, rotated rx 0 ry -90 rz 43.24 deg; joints [-4.11, 8.82, 14.191, 96.35, -104.596, 103.825, -773.241]
  MoveL 204 to (-51.17, 283.7, 120) mm, rotated rx 0 ry -90 rz 36.63 deg; joints [-4.389, 7.306, 17.275, 96.63, -104.165, 105.405, -766.632]
  MoveL 205 to (-47.33, 289.58, 110) mm, rotated rx 0 ry -90 rz 30.09 deg; joints [-4.669, 6.275, 19.381, 96.77, -103.788, 106.476, -760.094]
  MoveL 206 to (-42.85, 294.92, 100) mm, rotated rx 0 ry -90 rz 23.65 deg; joints [-4.949, 5.443, 21.088, 96.849, -103.435, 107.339, -753.654]
  MoveL 207 to (-37.86, 299.62, 90) mm, rotated rx 0 ry -90 rz 17.34 deg; joints [-5.229, 4.727, 22.562, 96.893, -103.096, 108.081, -747.341]
  MoveL 208 to (-32.46, 303.64, 80) mm, rotated rx 0 ry -90 rz 11.18 deg; joints [-5.509, 4.087, 23.88, 96.911, -102.768, 108.742, -741.181]
  MoveL 209 to (-26.8, 306.94, 70) mm, rotated rx 0 ry -90 rz 5.2 deg; joints [-5.79, 3.505, 25.084, 96.909, -102.448, 109.343, -735.202]
  MoveL 210 to (-21, 309.52, 60) mm, rotated rx 0 ry -90 rz -0.57 deg; joints [-6.071, 2.968, 26.198, 96.892, -102.134, 109.899, -729.431]
  MoveL 211 to (-15.19, 311.39, 50) mm, rotated rx 0 ry -90 rz -6.1 deg; joints [-6.352, 2.466, 27.24, 96.861, -101.826, 110.418, -723.896]
  MoveL 212 to (-9.5, 312.61, 40) mm, rotated rx 0 ry -90 rz -11.38 deg; joints [-6.634, 1.995, 28.221, 96.819, -101.523, 110.905, -718.624]
  MoveL 213 to (-4.03, 313.25, 30) mm, rotated rx 0 ry -90 rz -16.35 deg; joints [-6.916, 1.551, 29.147, 96.767, -101.225, 111.364, -713.645]
  MoveL 214 to (1.12, 313.37, 20) mm, rotated rx 0 ry -90 rz -21.01 deg; joints [-7.198, 1.132, 30.026, 96.705, -100.93, 111.799, -708.989]
  MoveL 215 to (5.87, 313.09, 10) mm, rotated rx 0 ry -90 rz -25.31 deg; joints [-7.481, 0.734, 30.859, 96.635, -100.64, 112.212, -704.685]
  MoveL 216 to (10.16, 312.5, 0) mm, rotated rx 0 ry -90 rz -29.23 deg; joints [-7.765, 0.357, 31.651, 96.557, -100.353, 112.603, -700.767]
  Set speed (1000.0 mm/s)
  MoveL 217 to (10.16, 312.5, 0) mm, rotated rx 0 ry -90 rz -29.23 deg; joints [-7.765, 0.357, 31.651, 96.557, -100.353, 112.603, -700.767]
  Set speed (1000.0 mm/s)
  MoveL 218 to (-37.62, 299.82, 0) mm, rotated rx 0 ry -90 rz 17.06 deg; joints [-7.759, 0.223, 31.945, 96.589, -100.339, 112.764, -747.061]
  MoveL 219 to (-37.62, 299.82, 0) mm, rotated rx 0 ry -90 rz 17.06 deg; joints [-7.759, 0.223, 31.945, 96.589, -100.339, 112.764, -747.061]
  Set speed (60.0 mm/s)
  MoveL 220 to (-40.85, 296.93, 10) mm, rotated rx 0 ry -90 rz 21.04 deg; joints [-7.474, 0.556, 31.247, 96.678, -100.621, 112.424, -751.039]
  MoveL 221 to (-44.15, 293.5, 20) mm, rotated rx 0 ry -90 rz 25.42 deg; joints [-7.19, 0.904, 30.521, 96.761, -100.906, 112.071, -755.425]
  MoveL 222 to (-47.39, 289.5, 30) mm, rotated rx 0 ry -90 rz 30.19 deg; joints [-6.905, 1.267, 29.765, 96.838, -101.194, 111.702, -760.19]
  MoveL 223 to (-50.45, 284.92, 40) mm, rotated rx 0 ry -90 rz 35.31 deg; joints [-6.621, 1.646, 28.975, 96.908, -101.486, 111.316, -765.308]
  MoveL 224 to (-53.21, 279.8, 50) mm, rotated rx 0 ry -90 rz 40.75 deg; joints [-6.337, 2.045, 28.146, 96.97, -101.781, 110.911, -770.751]
  MoveL 225 to (-55.55, 274.16, 60) mm, rotated rx 0 ry -90 rz 46.49 deg; joints [-6.054, 2.466, 27.273, 97.023, -102.079, 110.484, -776.493]
  MoveL 226 to (-57.35, 268.08, 70) mm, rotated rx 0 ry -90 rz 52.51 deg; joints [-5.771, 2.914, 26.347, 97.066, -102.383, 110.029, -782.507]
  MoveL 227 to (-58.51, 261.62, 80) mm, rotated rx 0 ry -90 rz 58.76 deg; joints [-5.488, 3.395, 25.355, 97.097, -102.691, 109.54, -788.765]
  MoveL 228 to (-58.95, 254.91, 90) mm, rotated rx 0 ry -90 rz 65.24 deg; joints [-5.205, 3.916, 24.28, 97.113, -103.006, 109.008, -795.24]
  MoveL 229 to (-58.6, 248.05, 100) mm, rotated rx 0 ry -90 rz 71.9 deg; joints [-4.923, 4.491, 23.097, 97.111, -103.329, 108.42, -801.902]
  MoveL 230 to (-57.44, 241.19, 110) mm, rotated rx 0 ry -90 rz 78.72 deg; joints [-4.642, 5.137, 21.769, 97.085, -103.661, 107.755, -808.721]
  MoveL 231 to (-55.46, 234.45, 120) mm, rotated rx 0 ry -90 rz 85.66 deg; joints [-4.361, 5.887, 20.23, 97.025, -104.007, 106.981, -815.664]
  MoveL 232 to (-52.68, 227.97, 130) mm, rotated rx 0 ry -90 rz 92.7 deg; joints [-4.081, 6.802, 18.358, 96.914, -104.374, 106.033, -822.696]
  MoveL 233 to (-49.15, 221.88, 140) mm, rotated rx 0 ry -90 rz 99.78 deg; joints [-3.802, 8.043, 15.826, 96.704, -104.779, 104.739, -829.78]
  MoveL 234 to (-44.74, 216.34, 149.94) mm, rotated rx 0 ry -90 rz 106.88 deg; joints [-3.524, 10.899, 10.028, 96.03, -105.361, 101.741, -836.877]
  MoveL 235 to (-37.8, 212.27, 159.24) mm, rotated rx 0 ry -90 rz 113.94 deg; joints [-3.247, 10.885, 10.028, 96.133, -105.62, 101.755, -843.944]
  MoveL 236 to (-30.59, 209.42, 168.5) mm, rotated rx 0 ry -90 rz 120.94 deg; joints [-2.971, 10.871, 10.028, 96.235, -105.878, 101.769, -850.939]
  MoveL 237 to (-29.38, 203.32, 180) mm, rotated rx 0 ry -90 rz 117.81 deg; joints [-2.2, 24.317, -17.489, 92.186, -107.67, 77.167, -857.814]
  MoveL 238 to (-23.62, 200.42, 190) mm, rotated rx 0 ry -90 rz 124.52 deg; joints [-1.919, 23.894, -16.67, 92.351, -107.933, 77.595, -864.525]
  MoveL 239 to (-17.8, 198.23, 200) mm, rotated rx 0 ry -90 rz 131.02 deg; joints [-1.64, 23.444, -15.796, 92.529, -108.191, 78.053, -871.023]
  MoveL 240 to (-12.04, 196.73, 210) mm, rotated rx 0 ry -90 rz 137.26 deg; joints [-1.362, 22.963, -14.862, 92.721, -108.445, 78.543, -877.262]
  MoveL 241 to (-6.46, 195.84, 220) mm, rotated rx 0 ry -90 rz 143.2 deg; joints [-1.085, 22.449, -13.862, 92.929, -108.695, 79.069, -883.197]
  MoveL 242 to (-1.16, 195.49, 230) mm, rotated rx 0 ry -90 rz 148.78 deg; joints [-0.81, 21.898, -12.791, 93.153, -108.939, 79.633, -888.782]
  MoveL 243 to (3.78, 195.6, 240) mm, rotated rx 0 ry -90 rz 153.97 deg; joints [-0.536, 21.307, -11.64, 93.396, -109.176, 80.242, -893.974]
  MoveL 244 to (8.28, 196.07, 250) mm, rotated rx 0 ry -90 rz 158.73 deg; joints [-0.263, 20.671, -10.398, 93.661, -109.407, 80.9, -898.733]
  MoveL 245 to (12.3, 196.78, 260) mm, rotated rx 0 ry -90 rz 163.02 deg; joints [0.008, 19.983, -9.05, 93.95, -109.63, 81.616, -903.017]
  MoveL 246 to (15.8, 197.64, 270) mm, rotated rx 0 ry -90 rz 166.79 deg; joints [0.279, 19.231, -7.578, 94.268, -109.843, 82.401, -906.788]
  MoveL 247 to (18.74, 198.54, 280) mm, rotated rx 0 ry -90 rz 170.01 deg; joints [0.548, 18.402, -5.948, 94.622, -110.044, 83.272, -910.01]
  MoveL 248 to (21.11, 199.39, 290) mm, rotated rx 0 ry -90 rz 172.64 deg; joints [0.817, 17.471, -4.111, 95.02, -110.229, 84.256, -912.645]
  Set speed (1000.0 mm/s)
  MoveL 249 to (21.11, 199.39, 290) mm, rotated rx 0 ry -90 rz 172.64 deg; joints [0.817, 17.471, -4.111, 95.02, -110.229, 84.256, -912.645]
  Set speed (1000.0 mm/s)
  MoveL 250 to (34.26, 188.12, 288.36) mm, rotated rx 0 ry -90 rz 177.69 deg; joints [0.617, 10.244, 10.028, 97.427, -109.288, 91.536, -917.692]
  MoveL 251 to (34.26, 188.12, 288.36) mm, rotated rx 0 ry -90 rz 177.69 deg; joints [0.617, 10.244, 10.028, 97.427, -109.288, 91.536, -917.692]
  Set speed (60.0 mm/s)
  MoveL 252 to (21.11, 199.39, 290) mm, rotated rx 0 ry -90 rz 172.64 deg; joints [0.817, 17.471, -4.111, 95.02, -110.229, 84.256, -912.645]
  Set speed (1000.0 mm/s)
  MoveL 253 to (21.11, 199.39, 290) mm, rotated rx 0 ry -90 rz 172.64 deg; joints [0.817, 17.471, -4.111, 95.02, -110.229, 84.256, -912.645]
  Set speed (1000.0 mm/s)
  MoveL 254 to (-55.59, 310.29, 0) mm, rotated rx 0 ry -90 rz 22.68 deg; joints [-7.877, 17.834, -4.128, 92.913, -101.773, 94.006, -752.681]
  MoveL 255 to (-55.59, 310.29, 0) mm, rotated rx 0 ry -90 rz 22.68 deg; joints [-7.877, 17.834, -4.128, 92.913, -101.773, 94.006, -752.681]
  Set speed (60.0 mm/s)
  MoveL 256 to (-37.62, 299.82, 0) mm, rotated rx 0 ry -90 rz 17.06 deg; joints [-7.759, 21.912, -11.889, 92.162, -102.051, 90.251, -747.061]
  Set speed (1000.0 mm/s)
  MoveL 257 to (-37.62, 299.82, 0) mm, rotated rx 0 ry -90 rz 17.06 deg; joints [-7.759, 21.912, -11.889, 92.162, -102.051, 90.251, -747.061]
  Set speed (1000.0 mm/s)
  MoveL 258 to (34.26, 188.12, 288.36) mm, rotated rx 0 ry -90 rz 177.69 deg; joints [0.617, 10.244, 10.028, 97.427, -109.288, 91.536, -917.692]
  MoveL 259 to (34.26, 188.12, 288.36) mm, rotated rx 0 ry -90 rz 177.69 deg; joints [0.617, 10.244, 10.028, 97.427, -109.288, 91.536, -917.692]
  Set speed (60.0 mm/s)
  MoveL 260 to (31.65, 183.43, 279.59) mm, rotated rx 0 ry -90 rz 175.11 deg; joints [0.351, 10.266, 10.028, 97.331, -109.037, 91.525, -915.112]
  MoveL 261 to (27.92, 180.74, 270) mm, rotated rx 0 ry -90 rz 171.96 deg; joints [0.084, 7.338, 15.99, 98.238, -108.38, 94.663, -911.958]
  MoveL 262 to (23.38, 179.17, 260) mm, rotated rx 0 ry -90 rz 168.27 deg; joints [-0.185, 5.635, 19.476, 98.694, -107.876, 96.481, -908.265]
  MoveL 263 to (18.11, 177.74, 250) mm, rotated rx 0 ry -90 rz 164.07 deg; joints [-0.454, 4.43, 21.954, 98.966, -107.441, 97.762, -904.071]
  MoveL 264 to (12.17, 176.57, 240) mm, rotated rx 0 ry -90 rz 159.41 deg; joints [-0.724, 3.455, 23.968, 99.15, -107.039, 98.797, -899.412]
  MoveL 265 to (5.61, 175.83, 230) mm, rotated rx 0 ry -90 rz 154.33 deg; joints [-0.995, 2.622, 25.694, 99.278, -106.659, 99.677, -894.325]
  MoveL 266 to (-1.49, 175.64, 220) mm, rotated rx 0 ry -90 rz 148.85 deg; joints [-1.268, 1.889, 27.215, 99.366, -106.296, 100.449, -888.851]
  MoveL 267 to (-9.03, 176.15, 210) mm, rotated rx 0 ry -90 rz 143.03 deg; joints [-1.542, 1.234, 28.579, 99.422, -105.945, 101.136, -883.03]
  MoveL 268 to (-16.88, 177.46, 200) mm, rotated rx 0 ry -90 rz 136.9 deg; joints [-1.817, 0.641, 29.815, 99.452, -105.604, 101.755, -876.902]
  MoveL 269 to (-24.89, 179.66, 190) mm, rotated rx 0 ry -90 rz 130.51 deg; joints [-2.093, 0.1, 30.945, 99.461, -105.273, 102.316, -870.512]
  MoveL 270 to (-32.91, 182.83, 180) mm, rotated rx 0 ry -90 rz 123.9 deg; joints [-2.371, -0.396, 31.982, 99.45, -104.95, 102.829, -863.901]
  MoveL 271 to (-40.75, 186.98, 170) mm, rotated rx 0 ry -90 rz 117.11 deg; joints [-2.65, -0.854, 32.94, 99.423, -104.634, 103.299, -857.113]
  MoveL 272 to (-48.24, 192.12, 160) mm, rotated rx 0 ry -90 rz 110.19 deg; joints [-2.931, -1.278, 33.828, 99.381, -104.325, 103.732, -850.193]
  MoveL 273 to (-55.2, 198.19, 150) mm, rotated rx 0 ry -90 rz 103.18 deg; joints [-3.212, -1.672, 34.654, 99.327, -104.021, 104.132, -843.183]
  MoveL 274 to (-61.48, 205.13, 140) mm, rotated rx 0 ry -90 rz 96.13 deg; joints [-3.495, -2.04, 35.426, 99.261, -103.723, 104.502, -836.127]
  MoveL 275 to (-66.92, 212.81, 130) mm, rotated rx 0 ry -90 rz 89.06 deg; joints [-3.779, -2.386, 36.15, 99.185, -103.429, 104.848, -829.064]
  MoveL 276 to (-71.41, 221.1, 120) mm, rotated rx 0 ry -90 rz 82.04 deg; joints [-4.063, -2.711, 36.832, 99.1, -103.139, 105.171, -822.035]
  MoveL 277 to (-74.87, 229.83, 110) mm, rotated rx 0 ry -90 rz 75.08 deg; joints [-4.349, -3.02, 37.478, 99.008, -102.853, 105.476, -815.078]
  MoveL 278 to (-77.24, 238.83, 100) mm, rotated rx 0 ry -90 rz 68.23 deg; joints [-4.635, -3.313, 38.094, 98.909, -102.57, 105.764, -808.229]
  MoveL 279 to (-74.4, 246.44, 88.88) mm, rotated rx 0 ry -90 rz 71.52 deg; joints [-5.345, 10.737, 10.028, 95.297, -103.684, 101.401, -801.522]
  MoveL 280 to (-76.57, 255.83, 79.39) mm, rotated rx 0 ry -90 rz 64.99 deg; joints [-5.625, 10.746, 10.028, 95.194, -103.423, 101.386, -794.991]
  MoveL 281 to (-77.56, 265.35, 69.87) mm, rotated rx 0 ry -90 rz 58.67 deg; joints [-5.905, 10.756, 10.028, 95.092, -103.161, 101.372, -788.666]
  MoveL 282 to (-76.35, 273.96, 60) mm, rotated rx 0 ry -90 rz 52.58 deg; joints [-6.186, 8.45, 14.709, 95.523, -102.682, 103.773, -782.579]
  MoveL 283 to (-73.92, 281.75, 50) mm, rotated rx 0 ry -90 rz 46.76 deg; joints [-6.467, 7.205, 17.244, 95.689, -102.3, 105.063, -776.759]
  MoveL 284 to (-70.87, 288.9, 40) mm, rotated rx 0 ry -90 rz 41.24 deg; joints [-6.748, 6.304, 19.085, 95.766, -101.952, 105.993, -771.235]
  MoveL 285 to (-67.34, 295.36, 30) mm, rotated rx 0 ry -90 rz 36.04 deg; joints [-7.03, 5.563, 20.603, 95.799, -101.621, 106.757, -766.036]
  MoveL 286 to (-63.51, 301.08, 20) mm, rotated rx 0 ry -90 rz 31.19 deg; joints [-7.312, 4.921, 21.923, 95.805, -101.302, 107.419, -761.192]
  MoveL 287 to (-59.54, 306.05, 10) mm, rotated rx 0 ry -90 rz 26.73 deg; joints [-7.594, 4.346, 23.105, 95.79, -100.99, 108.009, -756.73]
  MoveL 288 to (-55.59, 310.29, 0) mm, rotated rx 0 ry -90 rz 22.68 deg; joints [-7.877, 3.824, 24.184, 95.76, -100.685, 108.547, -752.681]
  Set speed (1000.0 mm/s)
  MoveL 289 to (-55.59, 310.29, 0) mm, rotated rx 0 ry -90 rz 22.68 deg; joints [-7.877, 3.824, 24.184, 95.76, -100.685, 108.547, -752.681]
  Set speed (1000.0 mm/s)
  MoveL 290 to (34.26, 188.12, 288.36) mm, rotated rx 0 ry -90 rz 177.69 deg; joints [0.617, 10.244, 10.028, 97.427, -109.288, 91.536, -917.692]
  MoveL 291 to (34.26, 188.12, 288.36) mm, rotated rx 0 ry -90 rz 177.69 deg; joints [0.617, 10.244, 10.028, 97.427, -109.288, 91.536, -917.692]
  Set speed (60.0 mm/s)
  MoveL 292 to (30.72, 204.12, 290) mm, rotated rx 0 ry -90 rz -176.2 deg; joints [0.813, 3.565, 23.982, 99.971, -108.363, 99.162, -923.801]
  Set speed (1000.0 mm/s)
  MoveL 293 to (30.72, 204.12, 290) mm, rotated rx 0 ry -90 rz -176.2 deg; joints [0.813, 3.565, 23.982, 99.971, -108.363, 99.162, -923.801]
  Set speed (1000.0 mm/s)
  MoveL 294 to (-55.59, 310.29, 0) mm, rotated rx 0 ry -90 rz 22.68 deg; joints [-7.877, 3.824, 24.184, 95.76, -100.685, 108.547, -752.681]
  MoveL 295 to (-55.59, 310.29, 0) mm, rotated rx 0 ry -90 rz 22.68 deg; joints [-7.877, 3.824, 24.184, 95.76, -100.685, 108.547, -752.681]
  Set speed (60.0 mm/s)
  MoveL 296 to (-45.21, 292.27, 0) mm, rotated rx 0 ry -90 rz 26.93 deg; joints [-7.756, 0.143, 32.12, 96.608, -100.331, 112.861, -756.927]
  Set speed (1000.0 mm/s)
  MoveL 297 to (-45.21, 292.27, 0) mm, rotated rx 0 ry -90 rz 26.93 deg; joints [-7.756, 0.143, 32.12, 96.608, -100.331, 112.861, -756.927]
  Set speed (1000.0 mm/s)
  MoveL 298 to (-55.59, 310.29, 0) mm, rotated rx 0 ry -90 rz 22.68 deg; joints [-7.877, 3.824, 24.184, 95.76, -100.685, 108.547, -752.681]
  MoveL 299 to (-55.59, 310.29, 0) mm, rotated rx 0 ry -90 rz 22.68 deg; joints [-7.877, 3.824, 24.184, 95.76, -100.685, 108.547, -752.681]
  Set speed (60.0 mm/s)
  MoveL 300 to (-59.54, 306.05, 10) mm, rotated rx 0 ry -90 rz 26.73 deg; joints [-7.594, 4.346, 23.105, 95.79, -100.99, 108.009, -756.73]
  MoveL 301 to (-63.51, 301.08, 20) mm, rotated rx 0 ry -90 rz 31.19 deg; joints [-7.312, 4.921, 21.923, 95.805, -101.302, 107.419, -761.192]
  MoveL 302 to (-67.34, 295.36, 30) mm, rotated rx 0 ry -90 rz 36.04 deg; joints [-7.03, 5.563, 20.603, 95.799, -101.621, 106.757, -766.036]
  MoveL 303 to (-70.87, 288.9, 40) mm, rotated rx 0 ry -90 rz 41.24 deg; joints [-6.748, 6.304, 19.085, 95.766, -101.952, 105.993, -771.235]
  MoveL 304 to (-73.92, 281.75, 50) mm, rotated rx 0 ry -90 rz 46.76 deg; joints [-6.467, 7.205, 17.244, 95.689, -102.3, 105.063, -776.759]
  MoveL 305 to (-76.35, 273.96, 60) mm, rotated rx 0 ry -90 rz 52.58 deg; joints [-6.186, 8.45, 14.709, 95.523, -102.682, 103.773, -782.579]
  MoveL 306 to (-77.56, 265.35, 69.87) mm, rotated rx 0 ry -90 rz 58.67 deg; joints [-5.905, 10.756, 10.028, 95.092, -103.161, 101.372, -788.666]
  MoveL 307 to (-76.57, 255.83, 79.39) mm, rotated rx 0 ry -90 rz 64.99 deg; joints [-5.625, 10.746, 10.028, 95.194, -103.423, 101.386, -794.991]
  MoveL 308 to (-74.4, 246.44, 88.88) mm, rotated rx 0 ry -90 rz 71.52 deg; joints [-5.345, 10.737, 10.028, 95.297, -103.684, 101.401, -801.522]
  MoveL 309 to (-77.24, 238.83, 100) mm, rotated rx 0 ry -90 rz 68.23 deg; joints [-4.635, 24.459, -18.038, 91.76, -105.266, 76.657, -808.229]
  MoveL 310 to (-74.87, 229.83, 110) mm, rotated rx 0 ry -90 rz 75.08 deg; joints [-4.349, 24.144, -17.423, 91.878, -105.541, 76.977, -815.078]
  MoveL 311 to (-71.41, 221.1, 120) mm, rotated rx 0 ry -90 rz 82.04 deg; joints [-4.063, 23.813, -16.776, 92.003, -105.814, 77.314, -822.035]
  MoveL 312 to (-66.92, 212.81, 130) mm, rotated rx 0 ry -90 rz 89.06 deg; joints [-3.779, 23.463, -16.094, 92.137, -106.084, 77.671, -829.064]
  MoveL 313 to (-61.48, 205.13, 140) mm, rotated rx 0 ry -90 rz 96.13 deg; joints [-3.495, 23.092, -15.37, 92.28, -106.351, 78.05, -836.127]
  MoveL 314 to (-55.2, 198.19, 150) mm, rotated rx 0 ry -90 rz 103.18 deg; joints [-3.212, 22.697, -14.598, 92.434, -106.616, 78.454, -843.183]
  MoveL 315 to (-48.24, 192.12, 160) mm, rotated rx 0 ry -90 rz 110.19 deg; joints [-2.931, 22.275, -13.772, 92.599, -106.876, 78.888, -850.193]
  MoveL 316 to (-40.75, 186.98, 170) mm, rotated rx 0 ry -90 rz 117.11 deg; joints [-2.65, 21.82, -12.885, 92.778, -107.133, 79.354, -857.113]
  MoveL 317 to (-32.91, 182.83, 180) mm, rotated rx 0 ry -90 rz 123.9 deg; joints [-2.371, 21.33, -11.927, 92.972, -107.384, 79.858, -863.901]
  MoveL 318 to (-24.89, 179.66, 190) mm, rotated rx 0 ry -90 rz 130.51 deg; joints [-2.093, 20.8, -10.889, 93.183, -107.631, 80.405, -870.512]
  MoveL 319 to (-16.88, 177.46, 200) mm, rotated rx 0 ry -90 rz 136.9 deg; joints [-1.817, 20.223, -9.76, 93.414, -107.87, 81.001, -876.902]
  MoveL 320 to (-9.03, 176.15, 210) mm, rotated rx 0 ry -90 rz 143.03 deg; joints [-1.542, 19.593, -8.523, 93.667, -108.103, 81.654, -883.03]
  MoveL 321 to (-1.49, 175.64, 220) mm, rotated rx 0 ry -90 rz 148.85 deg; joints [-1.268, 18.899, -7.16, 93.947, -108.326, 82.376, -888.851]
  MoveL 322 to (5.61, 175.83, 230) mm, rotated rx 0 ry -90 rz 154.33 deg; joints [-0.995, 18.126, -5.638, 94.259, -108.538, 83.183, -894.325]
  MoveL 323 to (12.17, 176.57, 240) mm, rotated rx 0 ry -90 rz 159.41 deg; joints [-0.724, 17.251, -3.913, 94.613, -108.736, 84.1, -899.412]
  MoveL 324 to (18.11, 177.74, 250) mm, rotated rx 0 ry -90 rz 164.07 deg; joints [-0.454, 16.234, -1.898, 95.024, -108.914, 85.173, -904.071]
  MoveL 325 to (23.38, 179.17, 260) mm, rotated rx 0 ry -90 rz 168.27 deg; joints [-0.185, 14.986, 0.58, 95.523, -109.06, 86.493, -908.265]
  MoveL 326 to (27.92, 180.74, 270) mm, rotated rx 0 ry -90 rz 171.96 deg; joints [0.084, 13.239, 4.066, 96.207, -109.138, 88.352, -911.958]
  MoveL 327 to (31.65, 183.43, 279.59) mm, rotated rx 0 ry -90 rz 175.11 deg; joints [0.351, 10.266, 10.028, 97.331, -109.037, 91.525, -915.112]
  MoveL 328 to (34.26, 188.12, 288.36) mm, rotated rx 0 ry -90 rz 177.69 deg; joints [0.617, 10.244, 10.028, 97.427, -109.288, 91.536, -917.692]
  Set speed (1000.0 mm/s)
  MoveL 329 to (34.26, 188.12, 288.36) mm, rotated rx 0 ry -90 rz 177.69 deg; joints [0.617, 10.244, 10.028, 97.427, -109.288, 91.536, -917.692]
  Set speed (1000.0 mm/s)
  MoveL 330 to (30.72, 204.12, 290) mm, rotated rx 0 ry -90 rz -176.2 deg; joints [0.813, 3.565, 23.982, 99.971, -108.363, 99.162, -923.801]
  MoveL 331 to (30.72, 204.12, 290) mm, rotated rx 0 ry -90 rz -176.2 deg; joints [0.813, 3.565, 23.982, 99.971, -108.363, 99.162, -923.801]
  Set speed (60.0 mm/s)
  MoveL 332 to (28.54, 202.85, 280) mm, rotated rx 0 ry -90 rz -178.82 deg; joints [0.545, 2.662, 25.854, 100.144, -107.961, 100.123, -921.184]
  MoveL 333 to (25.81, 201.43, 270) mm, rotated rx 0 ry -90 rz 177.98 deg; joints [0.276, 1.864, 27.513, 100.272, -107.576, 100.969, -917.983]
  MoveL 334 to (22.53, 199.96, 260) mm, rotated rx 0 ry -90 rz 174.23 deg; joints [0.006, 1.145, 29.013, 100.365, -107.206, 101.731, -914.232]
  MoveL 335 to (18.7, 198.53, 250) mm, rotated rx 0 ry -90 rz 169.97 deg; joints [-0.265, 0.489, 30.386, 100.431, -106.847, 102.423, -909.967]
  MoveL 336 to (14.35, 197.26, 240) mm, rotated rx 0 ry -90 rz 165.22 deg; joints [-0.537, -0.115, 31.653, 100.472, -106.498, 103.06, -905.225]
  MoveL 337 to (9.52, 196.26, 230) mm, rotated rx 0 ry -90 rz 160.04 deg; joints [-0.811, -0.675, 32.828, 100.493, -106.157, 103.647, -900.042]
  MoveL 338 to (4.24, 195.64, 220) mm, rotated rx 0 ry -90 rz 154.46 deg; joints [-1.085, -1.195, 33.923, 100.496, -105.825, 104.191, -894.46]
  MoveL 339 to (-1.41, 195.5, 210) mm, rotated rx 0 ry -90 rz 148.52 deg; joints [-1.361, -1.68, 34.945, 100.482, -105.5, 104.696, -888.518]
  MoveL 340 to (-7.35, 195.94, 200) mm, rotated rx 0 ry -90 rz 142.26 deg; joints [-1.638, -2.133, 35.902, 100.453, -105.181, 105.166, -882.261]
  MoveL 341 to (-13.47, 197.04, 190) mm, rotated rx 0 ry -90 rz 135.73 deg; joints [-1.917, -2.556, 36.797, 100.411, -104.869, 105.603, -875.734]
  MoveL 342 to (-19.65, 198.85, 180) mm, rotated rx 0 ry -90 rz 128.98 deg; joints [-2.196, -2.953, 37.637, 100.356, -104.562, 106.01, -868.982]
  MoveL 343 to (-22.28, 204.42, 168.61) mm, rotated rx 0 ry -90 rz 132.05 deg; joints [-2.967, 10.876, 10.028, 96.238, -105.881, 101.775, -862.053]
  MoveL 344 to (-29.95, 205.9, 159.38) mm, rotated rx 0 ry -90 rz 124.99 deg; joints [-3.243, 10.892, 10.028, 96.136, -105.624, 101.762, -854.993]
  MoveL 345 to (-37.3, 208.79, 150) mm, rotated rx 0 ry -90 rz 117.85 deg; joints [-3.519, 9.806, 12.251, 96.34, -105.244, 102.906, -847.85]
  MoveL 346 to (-42.45, 213.53, 140) mm, rotated rx 0 ry -90 rz 110.67 deg; joints [-3.797, 7.682, 16.571, 96.807, -104.739, 105.134, -840.67]
  MoveL 347 to (-47.02, 218.88, 130) mm, rotated rx 0 ry -90 rz 103.5 deg; joints [-4.076, 6.525, 18.935, 96.992, -104.343, 106.341, -833.496]
  MoveL 348 to (-50.93, 224.75, 120) mm, rotated rx 0 ry -90 rz 96.37 deg; joints [-4.356, 5.647, 20.735, 97.093, -103.98, 107.252, -826.37]
  MoveL 349 to (-54.1, 231.02, 110) mm, rotated rx 0 ry -90 rz 89.33 deg; joints [-4.636, 4.92, 22.227, 97.146, -103.636, 108.002, -819.332]
  MoveL 350 to (-56.49, 237.56, 100) mm, rotated rx 0 ry -90 rz 82.42 deg; joints [-4.918, 4.291, 23.521, 97.166, -103.306, 108.648, -812.418]
  MoveL 351 to (-58.06, 244.24, 90) mm, rotated rx 0 ry -90 rz 75.66 deg; joints [-5.2, 3.731, 24.673, 97.164, -102.985, 109.22, -805.663]
  MoveL 352 to (-58.85, 250.92, 80) mm, rotated rx 0 ry -90 rz 69.1 deg; joints [-5.482, 3.224, 25.72, 97.143, -102.672, 109.738, -799.1]
  MoveL 353 to (-58.87, 257.48, 70) mm, rotated rx 0 ry -90 rz 62.76 deg; joints [-5.765, 2.757, 26.685, 97.108, -102.365, 110.212, -792.759]
  MoveL 354 to (-58.2, 263.79, 60) mm, rotated rx 0 ry -90 rz 56.67 deg; joints [-6.049, 2.322, 27.585, 97.061, -102.064, 110.653, -786.668]
  MoveL 355 to (-56.92, 269.76, 50) mm, rotated rx 0 ry -90 rz 50.86 deg; joints [-6.332, 1.913, 28.432, 97.004, -101.766, 111.067, -780.857]
  MoveL 356 to (-55.13, 275.3, 40) mm, rotated rx 0 ry -90 rz 45.35 deg; joints [-6.616, 1.526, 29.235, 96.938, -101.473, 111.459, -775.351]
  MoveL 357 to (-52.95, 280.35, 30) mm, rotated rx 0 ry -90 rz 40.18 deg; joints [-6.901, 1.157, 30.002, 96.865, -101.183, 111.832, -770.178]
  MoveL 358 to (-50.48, 284.87, 20) mm, rotated rx 0 ry -90 rz 35.37 deg; joints [-7.186, 0.805, 30.736, 96.785, -100.896, 112.189, -765.365]
  MoveL 359 to (-47.86, 288.84, 10) mm, rotated rx 0 ry -90 rz 30.94 deg; joints [-7.471, 0.467, 31.441, 96.699, -100.612, 112.531, -760.939]
  MoveL 360 to (-45.21, 292.27, 0) mm, rotated rx 0 ry -90 rz 26.93 deg; joints [-7.756, 0.143, 32.12, 96.608, -100.331, 112.861, -756.927]
  Set speed (1000.0 mm/s)
  MoveL 361 to (-45.21, 292.27, 0) mm, rotated rx 0 ry -90 rz 26.93 deg; joints [-7.756, 0.143, 32.12, 96.608, -100.331, 112.861, -756.927]
  Set speed (1000.0 mm/s)
  MoveL 362 to (30.72, 204.12, 290) mm, rotated rx 0 ry -90 rz -176.2 deg; joints [0.813, 3.565, 23.982, 99.971, -108.363, 99.162, -923.801]
  MoveL 363 to (30.72, 204.12, 290) mm, rotated rx 0 ry -90 rz -176.2 deg; joints [0.813, 3.565, 23.982, 99.971, -108.363, 99.162, -923.801]
  Set speed (60.0 mm/s)
  MoveL 364 to (58.22, 245.2, 290) mm, rotated rx 0 ry -90 rz -124.72 deg; joints [0.781, 4.354, 22.312, 99.665, -108.485, 98.242, -975.284]
  Set speed (1000.0 mm/s)
  MoveL 365 to (58.22, 245.2, 290) mm, rotated rx 0 ry -90 rz -124.72 deg; joints [0.781, 4.354, 22.312, 99.665, -108.485, 98.242, -975.284]
  Set speed (1000.0 mm/s)
  MoveL 366 to (-45.21, 292.27, 0) mm, rotated rx 0 ry -90 rz 26.93 deg; joints [-7.756, 0.143, 32.12, 96.608, -100.331, 112.861, -1116.927]
  MoveL 367 to (-45.21, 292.27, 0) mm, rotated rx 0 ry -90 rz 26.93 deg; joints [-7.756, 0.143, 32.12, 96.608, -100.331, 112.861, -1116.927]
  Set speed (60.0 mm/s)
  MoveL 368 to (-58.12, 244.54, 0) mm, rotated rx 0 ry -90 rz 75.36 deg; joints [-7.735, -0.364, 33.232, 96.729, -100.279, 113.474, -1165.364]
  Set speed (1000.0 mm/s)
  MoveL 369 to (-58.12, 244.54, 0) mm, rotated rx 0 ry -90 rz 75.36 deg; joints [-7.735, -0.364, 33.232, 96.729, -100.279, 113.474, -1165.364]
  Set speed (1000.0 mm/s)
  MoveL 370 to (-45.21, 292.27, 0) mm, rotated rx 0 ry -90 rz 26.93 deg; joints [-7.756, 0.143, 32.12, 96.608, -100.331, 112.861, -1116.927]
  MoveL 371 to (-45.21, 292.27, 0) mm, rotated rx 0 ry -90 rz 26.93 deg; joints [-7.756, 0.143, 32.12, 96.608, -100.331, 112.861, -1116.927]
  Set speed (60.0 mm/s)
  MoveL 372 to (-47.86, 288.84, 10) mm, rotated rx 0 ry -90 rz 30.94 deg; joints [-7.471, 0.467, 31.441, 96.699, -100.612, 112.531, -1120.939]
  MoveL 373 to (-50.48, 284.87, 20) mm, rotated rx 0 ry -90 rz 35.37 deg; joints [-7.186, 0.805, 30.736, 96.785, -100.896, 112.189, -1125.365]
  MoveL 374 to (-52.95, 280.35, 30) mm, rotated rx 0 ry -90 rz 40.18 deg; joints [-6.901, 1.157, 30.002, 96.865, -101.183, 111.832, -1130.178]
  MoveL 375 to (-55.13, 275.3, 40) mm, rotated rx 0 ry -90 rz 45.35 deg; joints [-6.616, 1.526, 29.235, 96.938, -101.473, 111.459, -1135.351]
  MoveL 376 to (-56.92, 269.76, 50) mm, rotated rx 0 ry -90 rz 50.86 deg; joints [-6.332, 1.913, 28.432, 97.004, -101.766, 111.067, -1140.857]
  MoveL 377 to (-58.2, 263.79, 60) mm, rotated rx 0 ry -90 rz 56.67 deg; joints [-6.049, 2.322, 27.585, 97.061, -102.064, 110.653, -1146.668]
  MoveL 378 to (-58.87, 257.48, 70) mm, rotated rx 0 ry -90 rz 62.76 deg; joints [-5.765, 2.757, 26.685, 97.108, -102.365, 110.212, -1152.759]
  MoveL 379 to (-58.85, 250.92, 80) mm, rotated rx 0 ry -90 rz 69.1 deg; joints [-5.482, 3.224, 25.72, 97.143, -102.672, 109.738, -1159.1]
  MoveL 380 to (-58.06, 244.24, 90) mm, rotated rx 0 ry -90 rz 75.66 deg; joints [-5.2, 3.731, 24.673, 97.164, -102.985, 109.22, -1165.663]
  MoveL 381 to (-56.49, 237.56, 100) mm, rotated rx 0 ry -90 rz 82.42 deg; joints [-4.918, 4.291, 23.521, 97.166, -103.306, 108.648, -1172.418]
  MoveL 382 to (-54.1, 231.02, 110) mm, rotated rx 0 ry -90 rz 89.33 deg; joints [-4.636, 4.92, 22.227, 97.146, -103.636, 108.002, -1179.332]
  MoveL 383 to (-50.93, 224.75, 120) mm, rotated rx 0 ry -90 rz 96.37 deg; joints [-4.356, 5.647, 20.735, 97.093, -103.98, 107.252, -1186.37]
  MoveL 384 to (-47.02, 218.88, 130) mm, rotated rx 0 ry -90 rz 103.5 deg; joints [-4.076, 6.525, 18.935, 96.992, -104.343, 106.341, -1193.496]
  MoveL 385 to (-42.45, 213.53, 140) mm, rotated rx 0 ry -90 rz 110.67 deg; joints [-3.797, 7.682, 16.571, 96.807, -104.739, 105.134, -1200.67]
  MoveL 386 to (-37.3, 208.79, 150) mm, rotated rx 0 ry -90 rz 117.85 deg; joints [-3.519, 9.806, 12.251, 96.34, -105.244, 102.906, -1207.85]
  MoveL 387 to (-29.95, 205.9, 159.38) mm, rotated rx 0 ry -90 rz 124.99 deg; joints [-3.243, 10.892, 10.028, 96.136, -105.624, 101.762, -1214.993]
  MoveL 388 to (-22.28, 204.42, 168.61) mm, rotated rx 0 ry -90 rz 132.05 deg; joints [-2.967, 10.876, 10.028, 96.238, -105.881, 101.775, -1222.053]
  MoveL 389 to (-19.65, 198.85, 180) mm, rotated rx 0 ry -90 rz 128.98 deg; joints [-2.196, -2.953, 37.637, 100.356, -104.562, 106.01, -1228.982]
  MoveL 390 to (-13.47, 197.04, 190) mm, rotated rx 0 ry -90 rz 135.73 deg; joints [-1.917, -2.556, 36.797, 100.411, -104.869, 105.603, -1235.734]
  MoveL 391 to (-7.35, 195.94, 200) mm, rotated rx 0 ry -90 rz 142.26 deg; joints [-1.638, -2.133, 35.902, 100.453, -105.181, 105.166, -1242.261]
  MoveL 392 to (-1.41, 195.5, 210) mm, rotated rx 0 ry -90 rz 148.52 deg; joints [-1.361, -1.68, 34.945, 100.482, -105.5, 104.696, -1248.518]
  MoveL 393 to (4.24, 195.64, 220) mm, rotated rx 0 ry -90 rz 154.46 deg; joints [-1.085, -1.195, 33.923, 100.496, -105.825, 104.191, -1254.46]
  MoveL 394 to (9.52, 196.26, 230) mm, rotated rx 0 ry -90 rz 160.04 deg; joints [-0.811, -0.675, 32.828, 100.493, -106.157, 103.647, -1260.042]
  MoveL 395 to (14.35, 197.26, 240) mm, rotated rx 0 ry -90 rz 165.22 deg; joints [-0.537, -0.115, 31.653, 100.472, -106.498, 103.06, -1265.225]
  MoveL 396 to (18.7, 198.53, 250) mm, rotated rx 0 ry -90 rz 169.97 deg; joints [-0.265, 0.489, 30.386, 100.431, -106.847, 102.423, -1269.967]
  MoveL 397 to (22.53, 199.96, 260) mm, rotated rx 0 ry -90 rz 174.23 deg; joints [0.006, 1.145, 29.013, 100.365, -107.206, 101.731, -1274.232]
  MoveL 398 to (25.81, 201.43, 270) mm, rotated rx 0 ry -90 rz 177.98 deg; joints [0.276, 1.864, 27.513, 100.272, -107.576, 100.969, -1277.983]
  MoveL 399 to (28.54, 202.85, 280) mm, rotated rx 0 ry -90 rz -178.82 deg; joints [0.545, 2.662, 25.854, 100.144, -107.961, 100.123, -1281.184]
  MoveL 400 to (30.72, 204.12, 290) mm, rotated rx 0 ry -90 rz -176.2 deg; joints [0.813, 3.565, 23.982, 99.971, -108.363, 99.162, -1283.801]
  Set speed (1000.0 mm/s)
  MoveL 401 to (30.72, 204.12, 290) mm, rotated rx 0 ry -90 rz -176.2 deg; joints [0.813, 3.565, 23.982, 99.971, -108.363, 99.162, -1283.801]
  Set speed (1000.0 mm/s)
  MoveL 402 to (58.22, 245.2, 290) mm, rotated rx 0 ry -90 rz -124.72 deg; joints [0.781, 4.354, 22.312, 99.665, -108.485, 98.242, -1335.284]
  MoveL 403 to (58.22, 245.2, 290) mm, rotated rx 0 ry -90 rz -124.72 deg; joints [0.781, 4.354, 22.312, 99.665, -108.485, 98.242, -1335.284]
  Set speed (60.0 mm/s)
  MoveL 404 to (57.77, 242.72, 280) mm, rotated rx 0 ry -90 rz -127.19 deg; joints [0.514, 3.325, 24.441, 99.888, -108.064, 99.341, -1332.814]
  MoveL 405 to (57.08, 239.72, 270) mm, rotated rx 0 ry -90 rz -130.21 deg; joints [0.246, 2.434, 26.291, 100.052, -107.666, 100.291, -1329.788]
  MoveL 406 to (56.08, 236.26, 260) mm, rotated rx 0 ry -90 rz -133.77 deg; joints [-0.022, 1.639, 27.947, 100.175, -107.284, 101.136, -1326.235]
  MoveL 407 to (54.69, 232.42, 250) mm, rotated rx 0 ry -90 rz -137.82 deg; joints [-0.291, 0.917, 29.457, 100.267, -106.915, 101.904, -1322.184]
  MoveL 408 to (52.84, 228.29, 240) mm, rotated rx 0 ry -90 rz -142.34 deg; joints [-0.561, 0.252, 30.851, 100.332, -106.557, 102.61, -1317.664]
  MoveL 409 to (50.46, 223.96, 230) mm, rotated rx 0 ry -90 rz -147.29 deg; joints [-0.831, -0.364, 32.147, 100.376, -106.207, 103.265, -1312.705]
  MoveL 410 to (47.51, 219.54, 220) mm, rotated rx 0 ry -90 rz -152.66 deg; joints [-1.103, -0.94, 33.361, 100.4, -105.866, 103.875, -1307.337]
  MoveL 411 to (43.95, 215.15, 210) mm, rotated rx 0 ry -90 rz -158.41 deg; joints [-1.375, -1.479, 34.501, 100.407, -105.532, 104.446, -1301.59]
  MoveL 412 to (39.77, 210.92, 200) mm, rotated rx 0 ry -90 rz -164.5 deg; joints [-1.649, -1.986, 35.575, 100.399, -105.205, 104.981, -1295.499]
  MoveL 413 to (34.96, 206.97, 190) mm, rotated rx 0 ry -90 rz -170.9 deg; joints [-1.924, -2.462, 36.588, 100.376, -104.884, 105.484, -1289.096]
  MoveL 414 to (29.57, 203.44, 180) mm, rotated rx 0 ry -90 rz -177.58 deg; joints [-2.2, -2.911, 37.543, 100.341, -104.569, 105.957, -1282.421]
  MoveL 415 to (23.32, 204.97, 168.63) mm, rotated rx 0 ry -90 rz -174.49 deg; joints [-2.966, 10.877, 10.028, 96.239, -105.882, 101.776, -1275.511]
  MoveL 416 to (17.37, 199.72, 159.51) mm, rotated rx 0 ry -90 rz 178.41 deg; joints [-3.238, 10.898, 10.028, 96.14, -105.627, 101.769, -1268.409]
  MoveL 417 to (10.57, 196.44, 150) mm, rotated rx 0 ry -90 rz 171.16 deg; joints [-3.511, 8.771, 14.366, 96.634, -105.129, 104.019, -1261.159]
  MoveL 418 to (3.62, 195.59, 140) mm, rotated rx 0 ry -90 rz 163.81 deg; joints [-3.786, 7.011, 17.962, 96.999, -104.663, 105.874, -1253.808]
  MoveL 419 to (-3.42, 195.58, 130) mm, rotated rx 0 ry -90 rz 156.4 deg; joints [-4.061, 5.874, 20.296, 97.179, -104.268, 107.07, -1246.404]
  MoveL 420 to (-10.42, 196.41, 120) mm, rotated rx 0 ry -90 rz 148.99 deg; joints [-4.338, 4.987, 22.123, 97.281, -103.904, 107.999, -1238.993]
  MoveL 421 to (-17.25, 198.06, 110) mm, rotated rx 0 ry -90 rz 141.62 deg; joints [-4.617, 4.248, 23.648, 97.335, -103.559, 108.769, -1231.625]
  MoveL 422 to (-23.78, 200.49, 100) mm, rotated rx 0 ry -90 rz 134.35 deg; joints [-4.896, 3.611, 24.965, 97.356, -103.228, 109.43, -1224.346]
  MoveL 423 to (-29.89, 203.62, 90) mm, rotated rx 0 ry -90 rz 127.2 deg; joints [-5.176, 3.049, 26.129, 97.352, -102.908, 110.011, -1217.203]
  MoveL 424 to (-35.48, 207.36, 80) mm, rotated rx 0 ry -90 rz 120.24 deg; joints [-5.458, 2.545, 27.174, 97.328, -102.595, 110.529, -1210.238]
  MoveL 425 to (-40.49, 211.59, 70) mm, rotated rx 0 ry -90 rz 113.49 deg; joints [-5.74, 2.087, 28.124, 97.288, -102.29, 110.997, -1203.492]
  MoveL 426 to (-44.86, 216.19, 60) mm, rotated rx 0 ry -90 rz 107 deg; joints [-6.023, 1.667, 28.998, 97.234, -101.991, 111.425, -1197.004]
  MoveL 427 to (-48.58, 221.03, 50) mm, rotated rx 0 ry -90 rz 100.81 deg; joints [-6.307, 1.277, 29.808, 97.17, -101.696, 111.82, -1190.81]
  MoveL 428 to (-51.63, 225.99, 40) mm, rotated rx 0 ry -90 rz 94.94 deg; joints [-6.592, 0.913, 30.566, 97.096, -101.406, 112.189, -1184.943]
  MoveL 429 to (-54.06, 230.92, 30) mm, rotated rx 0 ry -90 rz 89.44 deg; joints [-6.877, 0.57, 31.281, 97.014, -101.12, 112.535, -1179.435]
  MoveL 430 to (-55.91, 235.73, 20) mm, rotated rx 0 ry -90 rz 84.32 deg; joints [-7.162, 0.244, 31.96, 96.925, -100.836, 112.862, -1174.317]
  MoveL 431 to (-57.23, 240.3, 10) mm, rotated rx 0 ry -90 rz 79.62 deg; joints [-7.448, -0.066, 32.609, 96.83, -100.556, 113.174, -1169.617]
  MoveL 432 to (-58.12, 244.54, 0) mm, rotated rx 0 ry -90 rz 75.36 deg; joints [-7.735, -0.364, 33.232, 96.729, -100.279, 113.474, -1165.364]
  Set speed (1000.0 mm/s)
  MoveL 433 to (-58.12, 244.54, 0) mm, rotated rx 0 ry -90 rz 75.36 deg; joints [-7.735, -0.364, 33.232, 96.729, -100.279, 113.474, -1165.364]
  Set speed (1000.0 mm/s)
  MoveL 434 to (58.22, 245.2, 290) mm, rotated rx 0 ry -90 rz -124.72 deg; joints [0.781, 4.354, 22.312, 99.665, -108.485, 98.242, -1335.284]
  MoveL 435 to (58.22, 245.2, 290) mm, rotated rx 0 ry -90 rz -124.72 deg; joints [0.781, 4.354, 22.312, 99.665, -108.485, 98.242, -1335.284]
  Set speed (60.0 mm/s)
  MoveL 436 to (78.63, 249.2, 290) mm, rotated rx 0 ry -90 rz -130.58 deg; joints [1.129, -3.542, 36.725, 101.942, -107.559, 95.033, -1339.419]
  Set speed (1000.0 mm/s)
  MoveL 437 to (78.63, 249.2, 290) mm, rotated rx 0 ry -90 rz -130.58 deg; joints [1.129, -3.542, 36.725, 101.942, -107.559, 95.033, -1339.419]
  Set speed (1000.0 mm/s)
  MoveL 438 to (-58.12, 244.54, 0) mm, rotated rx 0 ry -90 rz 75.36 deg; joints [-7.735, -0.364, 33.232, 96.729, -100.279, 113.474, -1165.364]
  MoveL 439 to (-58.12, 244.54, 0) mm, rotated rx 0 ry -90 rz 75.36 deg; joints [-7.735, -0.364, 33.232, 96.729, -100.279, 113.474, -1165.364]
  Set speed (60.0 mm/s)
  MoveL 440 to (-76.17, 234.21, 0) mm, rotated rx 0 ry -90 rz 81.71 deg; joints [-7.852, 2.89, 26.175, 95.97, -100.599, 109.619, -1171.709]
  Set speed (1000.0 mm/s)
  MoveL 441 to (-76.17, 234.21, 0) mm, rotated rx 0 ry -90 rz 81.71 deg; joints [-7.852, 2.89, 26.175, 95.97, -100.599, 109.619, -1171.709]
  Set speed (1000.0 mm/s)
  MoveL 442 to (-58.12, 244.54, 0) mm, rotated rx 0 ry -90 rz 75.36 deg; joints [-7.735, -0.364, 33.232, 96.729, -100.279, 113.474, -1165.364]
  MoveL 443 to (-58.12, 244.54, 0) mm, rotated rx 0 ry -90 rz 75.36 deg; joints [-7.735, -0.364, 33.232, 96.729, -100.279, 113.474, -1165.364]
  Set speed (60.0 mm/s)
  MoveL 444 to (-57.23, 240.3, 10) mm, rotated rx 0 ry -90 rz 79.62 deg; joints [-7.448, -0.066, 32.609, 96.83, -100.556, 113.174, -1169.617]
  MoveL 445 to (-55.91, 235.73, 20) mm, rotated rx 0 ry -90 rz 84.32 deg; joints [-7.162, 0.244, 31.96, 96.925, -100.836, 112.862, -1174.317]
  MoveL 446 to (-54.06, 230.92, 30) mm, rotated rx 0 ry -90 rz 89.44 deg; joints [-6.877, 0.57, 31.281, 97.014, -101.12, 112.535, -1179.435]
  MoveL 447 to (-51.63, 225.99, 40) mm, rotated rx 0 ry -90 rz 94.94 deg; joints [-6.592, 0.913, 30.566, 97.096, -101.406, 112.189, -1184.943]
  MoveL 448 to (-48.58, 221.03, 50) mm, rotated rx 0 ry -90 rz 100.81 deg; joints [-6.307, 1.277, 29.808, 97.17, -101.696, 111.82, -1190.81]
  MoveL 449 to (-44.86, 216.19, 60) mm, rotated rx 0 ry -90 rz 107 deg; joints [-6.023, 1.667, 28.998, 97.234, -101.991, 111.425, -1197.004]
  MoveL 450 to (-40.49, 211.59, 70) mm, rotated rx 0 ry -90 rz 113.49 deg; joints [-5.74, 2.087, 28.124, 97.288, -102.29, 110.997, -1203.492]
  MoveL 451 to (-35.48, 207.36, 80) mm, rotated rx 0 ry -90 rz 120.24 deg; joints [-5.458, 2.545, 27.174, 97.328, -102.595, 110.529, -1210.238]
  MoveL 452 to (-29.89, 203.62, 90) mm, rotated rx 0 ry -90 rz 127.2 deg; joints [-5.176, 3.049, 26.129, 97.352, -102.908, 110.011, -1217.203]
  MoveL 453 to (-23.78, 200.49, 100) mm, rotated rx 0 ry -90 rz 134.35 deg; joints [-4.896, 3.611, 24.965, 97.356, -103.228, 109.43, -1224.346]
  MoveL 454 to (-17.25, 198.06, 110) mm, rotated rx 0 ry -90 rz 141.62 deg; joints [-4.617, 4.248, 23.648, 97.335, -103.559, 108.769, -1231.625]
  MoveL 455 to (-10.42, 196.41, 120) mm, rotated rx 0 ry -90 rz 148.99 deg; joints [-4.338, 4.987, 22.123, 97.281, -103.904, 107.999, -1238.993]
  MoveL 456 to (-3.42, 195.58, 130) mm, rotated rx 0 ry -90 rz 156.4 deg; joints [-4.061, 5.874, 20.296, 97.179, -104.268, 107.07, -1246.404]
  MoveL 457 to (3.62, 195.59, 140) mm, rotated rx 0 ry -90 rz 163.81 deg; joints [-3.786, 7.011, 17.962, 96.999, -104.663, 105.874, -1253.808]
  MoveL 458 to (10.57, 196.44, 150) mm, rotated rx 0 ry -90 rz 171.16 deg; joints [-3.511, 8.771, 14.366, 96.634, -105.129, 104.019, -1261.159]
  MoveL 459 to (17.37, 199.72, 159.51) mm, rotated rx 0 ry -90 rz 178.41 deg; joints [-3.238, 10.898, 10.028, 96.14, -105.627, 101.769, -1268.409]
  MoveL 460 to (23.32, 204.97, 168.63) mm, rotated rx 0 ry -90 rz -174.49 deg; joints [-2.966, 10.877, 10.028, 96.239, -105.882, 101.776, -1275.511]
  MoveL 461 to (29.57, 203.44, 180) mm, rotated rx 0 ry -90 rz -177.58 deg; joints [-2.2, 24.315, -17.487, 92.186, -107.67, 77.168, -1282.421]
  MoveL 462 to (34.96, 206.97, 190) mm, rotated rx 0 ry -90 rz -170.9 deg; joints [-1.924, 23.82, -16.532, 92.371, -107.925, 77.662, -1289.096]
  MoveL 463 to (39.77, 210.92, 200) mm, rotated rx 0 ry -90 rz -164.5 deg; joints [-1.649, 23.295, -15.519, 92.57, -108.176, 78.187, -1295.499]
  MoveL 464 to (43.95, 215.15, 210) mm, rotated rx 0 ry -90 rz -158.41 deg; joints [-1.375, 22.739, -14.446, 92.783, -108.423, 78.745, -1301.59]
  MoveL 465 to (47.51, 219.54, 220) mm, rotated rx 0 ry -90 rz -152.66 deg; joints [-1.103, 22.151, -13.305, 93.013, -108.664, 79.341, -1307.337]
  MoveL 466 to (50.46, 223.96, 230) mm, rotated rx 0 ry -90 rz -147.29 deg; joints [-0.831, 21.525, -12.092, 93.261, -108.899, 79.977, -1312.705]
  MoveL 467 to (52.84, 228.29, 240) mm, rotated rx 0 ry -90 rz -142.34 deg; joints [-0.561, 20.859, -10.795, 93.529, -109.128, 80.659, -1317.664]
  MoveL 468 to (54.69, 232.42, 250) mm, rotated rx 0 ry -90 rz -137.82 deg; joints [-0.291, 20.144, -9.401, 93.82, -109.35, 81.395, -1322.184]
  MoveL 469 to (56.08, 236.26, 260) mm, rotated rx 0 ry -90 rz -133.77 deg; joints [-0.022, 19.373, -7.891, 94.139, -109.562, 82.195, -1326.235]
  MoveL 470 to (57.08, 239.72, 270) mm, rotated rx 0 ry -90 rz -130.21 deg; joints [0.246, 18.528, -6.235, 94.49, -109.762, 83.076, -1329.788]
  MoveL 471 to (57.77, 242.72, 280) mm, rotated rx 0 ry -90 rz -127.19 deg; joints [0.514, 17.589, -4.385, 94.885, -109.948, 84.063, -1332.814]
  MoveL 472 to (58.22, 245.2, 290) mm, rotated rx 0 ry -90 rz -124.72 deg; joints [0.781, 16.511, -2.256, 95.338, -110.113, 85.202, -1335.284]
  Set speed (1000.0 mm/s)
  MoveL 473 to (58.22, 245.2, 290) mm, rotated rx 0 ry -90 rz -124.72 deg; joints [0.781, 16.511, -2.256, 95.338, -110.113, 85.202, -1335.284]
  Set speed (1000.0 mm/s)
  MoveL 474 to (78.63, 249.2, 290) mm, rotated rx 0 ry -90 rz -130.58 deg; joints [1.129, 22.875, -16.669, 92.392, -110.999, 66.65, -1339.419]
  MoveL 475 to (78.63, 249.2, 290) mm, rotated rx 0 ry -90 rz -130.58 deg; joints [1.129, 22.875, -16.669, 92.392, -110.999, 66.65, -1339.419]
  Set speed (60.0 mm/s)
  MoveL 476 to (74.53, 247.53, 278.49) mm, rotated rx 0 ry -90 rz -123.04 deg; joints [0.315, 10.224, 10.028, 97.303, -109.009, 91.477, -1336.964]
  MoveL 477 to (77.08, 242.12, 269.72) mm, rotated rx 0 ry -90 rz -126.04 deg; joints [0.049, 10.248, 10.028, 97.208, -108.759, 91.468, -1333.959]
  MoveL 478 to (76.86, 237.05, 260) mm, rotated rx 0 ry -90 rz -129.57 deg; joints [-0.217, 13.516, 3.471, 95.999, -108.887, 87.986, -1330.435]
  MoveL 479 to (75.48, 231.77, 250) mm, rotated rx 0 ry -90 rz -133.58 deg; joints [-0.483, 15.215, 0.087, 95.344, -108.798, 86.187, -1326.422]
  MoveL 480 to (73.51, 226.04, 240) mm, rotated rx 0 ry -90 rz -138.05 deg; joints [-0.751, 16.468, -2.398, 94.853, -108.65, 84.868, -1321.95]
  MoveL 481 to (70.88, 219.99, 230) mm, rotated rx 0 ry -90 rz -142.95 deg; joints [-1.019, 17.508, -4.45, 94.444, -108.472, 83.781, -1317.052]
  MoveL 482 to (67.49, 213.75, 220) mm, rotated rx 0 ry -90 rz -148.24 deg; joints [-1.288, 18.413, -6.231, 94.088, -108.275, 82.84, -1311.756]
  MoveL 483 to (63.28, 207.47, 210) mm, rotated rx 0 ry -90 rz -153.9 deg; joints [-1.558, 19.223, -7.819, 93.772, -108.065, 82.004, -1306.097]
  MoveL 484 to (58.22, 201.33, 200) mm, rotated rx 0 ry -90 rz -159.89 deg; joints [-1.829, 19.958, -9.257, 93.488, -107.844, 81.249, -1300.107]
  MoveL 485 to (52.31, 195.49, 190) mm, rotated rx 0 ry -90 rz -166.18 deg; joints [-2.102, 20.633, -10.574, 93.229, -107.614, 80.559, -1293.819]
  MoveL 486 to (45.56, 190.13, 180) mm, rotated rx 0 ry -90 rz -172.73 deg; joints [-2.375, 21.257, -11.789, 92.992, -107.377, 79.926, -1287.271]
  MoveL 487 to (38.04, 185.42, 170) mm, rotated rx 0 ry -90 rz -179.5 deg; joints [-2.649, 21.835, -12.913, 92.774, -107.134, 79.341, -1280.5]
  MoveL 488 to (29.85, 181.5, 160) mm, rotated rx 0 ry -90 rz 173.54 deg; joints [-2.925, 22.373, -13.957, 92.574, -106.885, 78.799, -1273.545]
  MoveL 489 to (21.11, 178.51, 150) mm, rotated rx 0 ry -90 rz 166.45 deg; joints [-3.203, 22.874, -14.928, 92.39, -106.631, 78.295, -1266.447]
  MoveL 490 to (11.96, 176.54, 140) mm, rotated rx 0 ry -90 rz 159.25 deg; joints [-3.481, 23.342, -15.834, 92.219, -106.373, 77.828, -1259.249]
  MoveL 491 to (2.59, 175.67, 130) mm, rotated rx 0 ry -90 rz 151.99 deg; joints [-3.761, 23.778, -16.678, 92.062, -106.111, 77.392, -1251.995]
  MoveL 492 to (-6.83, 175.92, 120) mm, rotated rx 0 ry -90 rz 144.73 deg; joints [-4.042, 24.186, -17.466, 91.916, -105.845, 76.986, -1244.728]
  MoveL 493 to (-12.97, 182.04, 108.48) mm, rotated rx 0 ry -90 rz 147.49 deg; joints [-4.764, 10.752, 10.028, 95.52, -104.223, 101.469, -1237.494]
  MoveL 494 to (-22.91, 182.28, 99.12) mm, rotated rx 0 ry -90 rz 140.34 deg; joints [-5.04, 10.767, 10.028, 95.419, -103.965, 101.459, -1230.336]
  MoveL 495 to (-32.8, 183.9, 89.72) mm, rotated rx 0 ry -90 rz 133.3 deg; joints [-5.318, 10.781, 10.028, 95.318, -103.705, 101.448, -1223.298]
  MoveL 496 to (-41.52, 187.45, 80) mm, rotated rx 0 ry -90 rz 126.42 deg; joints [-5.597, 12.838, 5.896, 94.715, -103.625, 99.298, -1216.42]
  MoveL 497 to (-48.7, 192.48, 70) mm, rotated rx 0 ry -90 rz 119.74 deg; joints [-5.876, 14.329, 2.909, 94.264, -103.477, 97.742, -1209.745]
  MoveL 498 to (-55.08, 198.08, 60) mm, rotated rx 0 ry -90 rz 113.31 deg; joints [-6.157, 15.329, 0.912, 93.942, -103.281, 96.7, -1203.31]
  MoveL 499 to (-60.61, 204.07, 50) mm, rotated rx 0 ry -90 rz 107.15 deg; joints [-6.438, 16.124, -0.673, 93.677, -103.063, 95.872, -1197.152]
  MoveL 500 to (-65.29, 210.3, 40) mm, rotated rx 0 ry -90 rz 101.31 deg; joints [-6.72, 16.798, -2.014, 93.447, -102.833, 95.172, -1191.307]
  MoveL 501 to (-69.12, 216.58, 30) mm, rotated rx 0 ry -90 rz 95.81 deg; joints [-7.002, 17.391, -3.192, 93.241, -102.594, 94.557, -1185.808]
  MoveL 502 to (-72.16, 222.75, 20) mm, rotated rx 0 ry -90 rz 90.69 deg; joints [-7.285, 17.925, -4.251, 93.053, -102.349, 94.005, -1180.687]
  MoveL 503 to (-74.48, 228.68, 10) mm, rotated rx 0 ry -90 rz 85.98 deg; joints [-7.568, 18.415, -5.22, 92.881, -102.099, 93.5, -1175.978]
  MoveL 504 to (-76.17, 234.21, 0) mm, rotated rx 0 ry -90 rz 81.71 deg; joints [-7.852, 18.869, -6.119, 92.72, -101.844, 93.033, -1171.709]
  Set speed (1000.0 mm/s)
  MoveL 505 to (-76.17, 234.21, 0) mm, rotated rx 0 ry -90 rz 81.71 deg; joints [-7.852, 18.869, -6.119, 92.72, -101.844, 93.033, -1171.709]
  Set speed (1000.0 mm/s)
  MoveL 506 to (78.63, 249.2, 290) mm, rotated rx 0 ry -90 rz -130.58 deg; joints [1.129, 22.875, -16.669, 92.392, -110.999, 66.65, -1339.419]
  MoveL 507 to (78.63, 249.2, 290) mm, rotated rx 0 ry -90 rz -130.58 deg; joints [1.129, 22.875, -16.669, 92.392, -110.999, 66.65, -1339.419]
  Set speed (60.0 mm/s)
  MoveL 508 to (58.93, 255.88, 290) mm, rotated rx 0 ry -90 rz -114.31 deg; joints [0.773, 16.276, -1.8, 95.417, -110.084, 85.436, -1345.694]
  Set speed (1000.0 mm/s)
  MoveL 509 to (58.93, 255.88, 290) mm, rotated rx 0 ry -90 rz -114.31 deg; joints [0.773, 16.276, -1.8, 95.417, -110.084, 85.436, -1345.694]
  Set speed (1000.0 mm/s)
  MoveL 510 to (-76.17, 234.21, 0) mm, rotated rx 0 ry -90 rz 81.71 deg; joints [-7.852, 18.869, -6.119, 92.72, -101.844, 93.033, -1171.709]
  MoveL 511 to (-76.17, 234.21, 0) mm, rotated rx 0 ry -90 rz 81.71 deg; joints [-7.852, 18.869, -6.119, 92.72, -101.844, 93.033, -1171.709]
  Set speed (60.0 mm/s)
  MoveL 512 to (-55.37, 234.2, 0) mm, rotated rx 0 ry -90 rz 85.93 deg; joints [-7.73, 22.728, -13.419, 92.015, -102.106, 89.523, -1175.929]
  Set speed (1000.0 mm/s)
  MoveL 513 to (-55.37, 234.2, 0) mm, rotated rx 0 ry -90 rz 85.93 deg; joints [-7.73, 22.728, -13.419, 92.015, -102.106, 89.523, -1175.929]
  Set speed (1000.0 mm/s)
  MoveL 514 to (-76.17, 234.21, 0) mm, rotated rx 0 ry -90 rz 81.71 deg; joints [-7.852, 18.869, -6.119, 92.72, -101.844, 93.033, -1171.709]
  MoveL 515 to (-76.17, 234.21, 0) mm, rotated rx 0 ry -90 rz 81.71 deg; joints [-7.852, 18.869, -6.119, 92.72, -101.844, 93.033, -1171.709]
  Set speed (60.0 mm/s)
  MoveL 516 to (-74.48, 228.68, 10) mm, rotated rx 0 ry -90 rz 85.98 deg; joints [-7.568, 18.415, -5.22, 92.881, -102.099, 93.5, -1175.978]
  MoveL 517 to (-72.16, 222.75, 20) mm, rotated rx 0 ry -90 rz 90.69 deg; joints [-7.285, 17.925, -4.251, 93.053, -102.349, 94.005, -1180.687]
  MoveL 518 to (-69.12, 216.58, 30) mm, rotated rx 0 ry -90 rz 95.81 deg; joints [-7.002, 17.391, -3.192, 93.241, -102.594, 94.557, -1185.808]
  MoveL 519 to (-65.29, 210.3, 40) mm, rotated rx 0 ry -90 rz 101.31 deg; joints [-6.72, 16.798, -2.014, 93.447, -102.833, 95.172, -1191.307]
  MoveL 520 to (-60.61, 204.07, 50) mm, rotated rx 0 ry -90 rz 107.15 deg; joints [-6.438, 16.124, -0.673, 93.677, -103.063, 95.872, -1197.152]
  MoveL 521 to (-55.08, 198.08, 60) mm, rotated rx 0 ry -90 rz 113.31 deg; joints [-6.157, 15.329, 0.912, 93.942, -103.281, 96.7, -1203.31]
  MoveL 522 to (-48.7, 192.48, 70) mm, rotated rx 0 ry -90 rz 119.74 deg; joints [-5.876, 14.329, 2.909, 94.264, -103.477, 97.742, -1209.745]
  MoveL 523 to (-41.52, 187.45, 80) mm, rotated rx 0 ry -90 rz 126.42 deg; joints [-5.597, 12.838, 5.896, 94.715, -103.625, 99.298, -1216.42]
  MoveL 524 to (-32.8, 183.9, 89.72) mm, rotated rx 0 ry -90 rz 133.3 deg; joints [-5.318, 10.781, 10.028, 95.318, -103.705, 101.448, -1223.298]
  MoveL 525 to (-22.91, 182.28, 99.12) mm, rotated rx 0 ry -90 rz 140.34 deg; joints [-5.04, 10.767, 10.028, 95.419, -103.965, 101.459, -1230.336]
  MoveL 526 to (-12.97, 182.04, 108.48) mm, rotated rx 0 ry -90 rz 147.49 deg; joints [-4.764, 10.752, 10.028, 95.52, -104.223, 101.469, -1237.494]
  MoveL 527 to (-6.83, 175.92, 120) mm, rotated rx 0 ry -90 rz 144.73 deg; joints [-4.042, -3.021, 37.522, 99.2, -103.095, 105.56, -1244.728]
  MoveL 528 to (2.59, 175.67, 130) mm, rotated rx 0 ry -90 rz 151.99 deg; joints [-3.761, -2.648, 36.734, 99.271, -103.391, 105.176, -1251.995]
  MoveL 529 to (11.96, 176.54, 140) mm, rotated rx 0 ry -90 rz 159.25 deg; joints [-3.481, -2.25, 35.889, 99.33, -103.693, 104.763, -1259.249]
  MoveL 530 to (21.11, 178.51, 150) mm, rotated rx 0 ry -90 rz 166.45 deg; joints [-3.203, -1.821, 34.984, 99.377, -104, 104.317, -1266.447]
  MoveL 531 to (29.85, 181.5, 160) mm, rotated rx 0 ry -90 rz 173.54 deg; joints [-2.925, -1.362, 34.013, 99.409, -104.313, 103.835, -1273.545]
  MoveL 532 to (38.04, 185.42, 170) mm, rotated rx 0 ry -90 rz -179.5 deg; joints [-2.649, -0.867, 32.969, 99.427, -104.633, 103.315, -1280.5]
  MoveL 533 to (45.56, 190.13, 180) mm, rotated rx 0 ry -90 rz -172.73 deg; joints [-2.375, -0.333, 31.844, 99.428, -104.96, 102.752, -1287.271]
  MoveL 534 to (52.31, 195.49, 190) mm, rotated rx 0 ry -90 rz -166.18 deg; joints [-2.102, 0.245, 30.63, 99.41, -105.294, 102.141, -1293.819]
  MoveL 535 to (58.22, 201.33, 200) mm, rotated rx 0 ry -90 rz -159.89 deg; joints [-1.829, 0.873, 29.313, 99.371, -105.638, 101.476, -1300.107]
  MoveL 536 to (63.28, 207.47, 210) mm, rotated rx 0 ry -90 rz -153.9 deg; joints [-1.558, 1.561, 27.875, 99.307, -105.992, 100.746, -1306.097]
  MoveL 537 to (67.49, 213.75, 220) mm, rotated rx 0 ry -90 rz -148.24 deg; joints [-1.288, 2.323, 26.287, 99.212, -106.358, 99.936, -1311.756]
  MoveL 538 to (70.88, 219.99, 230) mm, rotated rx 0 ry -90 rz -142.95 deg; joints [-1.019, 3.18, 24.506, 99.079, -106.739, 99.024, -1317.052]
  MoveL 539 to (73.51, 226.04, 240) mm, rotated rx 0 ry -90 rz -138.05 deg; joints [-0.751, 4.171, 22.453, 98.894, -107.141, 97.967, -1321.95]
  MoveL 540 to (75.48, 231.77, 250) mm, rotated rx 0 ry -90 rz -133.58 deg; joints [-0.483, 5.376, 19.969, 98.628, -107.573, 96.681, -1326.422]
  MoveL 541 to (76.86, 237.05, 260) mm, rotated rx 0 ry -90 rz -129.57 deg; joints [-0.217, 7.027, 16.584, 98.198, -108.067, 94.917, -1330.435]
  MoveL 542 to (77.08, 242.12, 269.72) mm, rotated rx 0 ry -90 rz -126.04 deg; joints [0.049, 10.248, 10.028, 97.208, -108.759, 91.468, -1333.959]
  MoveL 543 to (74.53, 247.53, 278.49) mm, rotated rx 0 ry -90 rz -123.04 deg; joints [0.315, 10.224, 10.028, 97.303, -109.009, 91.477, -1336.964]
  MoveL 544 to (78.63, 249.2, 290) mm, rotated rx 0 ry -90 rz -130.58 deg; joints [1.129, -3.542, 36.725, 101.942, -107.559, 95.033, -1339.419]
  Set speed (1000.0 mm/s)
  MoveL 545 to (78.63, 249.2, 290) mm, rotated rx 0 ry -90 rz -130.58 deg; joints [1.129, -3.542, 36.725, 101.942, -107.559, 95.033, -1339.419]
  Set speed (1000.0 mm/s)
  MoveL 546 to (58.93, 255.88, 290) mm, rotated rx 0 ry -90 rz -114.31 deg; joints [0.773, 4.57, 21.856, 99.582, -108.518, 97.992, -1345.694]
  MoveL 547 to (58.93, 255.88, 290) mm, rotated rx 0 ry -90 rz -114.31 deg; joints [0.773, 4.57, 21.856, 99.582, -108.518, 97.992, -1345.694]
  Set speed (60.0 mm/s)
  MoveL 548 to (58.94, 253.36, 280) mm, rotated rx 0 ry -90 rz -116.74 deg; joints [0.506, 3.507, 24.053, 99.817, -108.092, 99.127, -1343.258]
  MoveL 549 to (58.8, 250.28, 270) mm, rotated rx 0 ry -90 rz -119.73 deg; joints [0.238, 2.594, 25.949, 99.991, -107.691, 100.101, -1340.274]
  MoveL 550 to (58.44, 246.7, 260) mm, rotated rx 0 ry -90 rz -123.23 deg; joints [-0.03, 1.782, 27.639, 100.121, -107.307, 100.965, -1336.77]
  MoveL 551 to (57.77, 242.68, 250) mm, rotated rx 0 ry -90 rz -127.23 deg; joints [-0.299, 1.047, 29.176, 100.217, -106.935, 101.748, -1332.774]
  MoveL 552 to (56.69, 238.28, 240) mm, rotated rx 0 ry -90 rz -131.68 deg; joints [-0.568, 0.37, 30.593, 100.287, -106.575, 102.466, -1328.316]
  MoveL 553 to (55.14, 233.59, 230) mm, rotated rx 0 ry -90 rz -136.58 deg; joints [-0.838, -0.257, 31.912, 100.335, -106.224, 103.133, -1323.424]
  MoveL 554 to (53.04, 228.71, 220) mm, rotated rx 0 ry -90 rz -141.87 deg; joints [-1.11, -0.842, 33.147, 100.363, -105.881, 103.754, -1318.126]
  MoveL 555 to (50.33, 223.75, 210) mm, rotated rx 0 ry -90 rz -147.55 deg; joints [-1.382, -1.392, 34.309, 100.375, -105.546, 104.337, -1312.453]
  MoveL 556 to (46.98, 218.83, 200) mm, rotated rx 0 ry -90 rz -153.57 deg; joints [-1.655, -1.908, 35.404, 100.37, -105.217, 104.884, -1306.434]
  MoveL 557 to (42.97, 214.08, 190) mm, rotated rx 0 ry -90 rz -159.9 deg; joints [-1.929, -2.395, 36.438, 100.352, -104.894, 105.4, -1300.103]
  MoveL 558 to (38.31, 209.62, 180) mm, rotated rx 0 ry -90 rz -166.51 deg; joints [-2.204, -2.855, 37.416, 100.32, -104.578, 105.885, -1293.494]
  MoveL 559 to (31.73, 210.33, 168.53) mm, rotated rx 0 ry -90 rz -163.36 deg; joints [-2.97, 10.872, 10.028, 96.236, -105.879, 101.771, -1286.645]
  MoveL 560 to (26.91, 204.04, 159.43) mm, rotated rx 0 ry -90 rz -170.41 deg; joints [-3.241, 10.894, 10.028, 96.138, -105.625, 101.765, -1279.594]
  MoveL 561 to (20.88, 199.3, 150) mm, rotated rx 0 ry -90 rz -177.62 deg; joints [-3.513, 8.962, 13.974, 96.579, -105.151, 103.813, -1272.384]
  MoveL 562 to (14.2, 197.22, 140) mm, rotated rx 0 ry -90 rz 175.06 deg; joints [-3.787, 7.067, 17.844, 96.983, -104.669, 105.812, -1265.059]
  MoveL 563 to (7.28, 195.93, 130) mm, rotated rx 0 ry -90 rz 167.67 deg; joints [-4.062, 5.883, 20.277, 97.176, -104.269, 107.059, -1257.666]
  MoveL 564 to (0.24, 195.48, 120) mm, rotated rx 0 ry -90 rz 160.25 deg; joints [-4.338, 4.966, 22.167, 97.287, -103.902, 108.022, -1250.252]
  MoveL 565 to (-6.77, 195.87, 110) mm, rotated rx 0 ry -90 rz 152.87 deg; joints [-4.615, 4.205, 23.739, 97.347, -103.554, 108.818, -1242.866]
  MoveL 566 to (-13.63, 197.08, 100) mm, rotated rx 0 ry -90 rz 145.55 deg; joints [-4.894, 3.55, 25.095, 97.373, -103.221, 109.501, -1235.555]
  MoveL 567 to (-20.21, 199.05, 90) mm, rotated rx 0 ry -90 rz 138.37 deg; joints [-5.174, 2.974, 26.29, 97.373, -102.899, 110.098, -1228.366]
  MoveL 568 to (-26.38, 201.72, 80) mm, rotated rx 0 ry -90 rz 131.35 deg; joints [-5.455, 2.459, 27.36, 97.352, -102.585, 110.63, -1221.346]
  MoveL 569 to (-32.08, 204.97, 70) mm, rotated rx 0 ry -90 rz 124.54 deg; joints [-5.737, 1.992, 28.33, 97.314, -102.279, 111.11, -1214.536]
  MoveL 570 to (-37.21, 208.71, 60) mm, rotated rx 0 ry -90 rz 117.98 deg; joints [-6.019, 1.565, 29.218, 97.261, -101.979, 111.546, -1207.979]
  MoveL 571 to (-41.73, 212.8, 50) mm, rotated rx 0 ry -90 rz 111.71 deg; joints [-6.303, 1.171, 30.04, 97.198, -101.684, 111.948, -1201.712]
  MoveL 572 to (-45.64, 217.12, 40) mm, rotated rx 0 ry -90 rz 105.77 deg; joints [-6.587, 0.803, 30.805, 97.124, -101.394, 112.32, -1195.772]
  MoveL 573 to (-48.92, 221.54, 30) mm, rotated rx 0 ry -90 rz 100.19 deg; joints [-6.872, 0.458, 31.525, 97.042, -101.107, 112.669, -1190.192]
  MoveL 574 to (-51.6, 225.93, 20) mm, rotated rx 0 ry -90 rz 95 deg; joints [-7.158, 0.132, 32.206, 96.953, -100.824, 112.997, -1185.005]
  MoveL 575 to (-53.73, 230.19, 10) mm, rotated rx 0 ry -90 rz 90.24 deg; joints [-7.443, -0.178, 32.854, 96.857, -100.544, 113.31, -1180.24]
  MoveL 576 to (-55.37, 234.2, 0) mm, rotated rx 0 ry -90 rz 85.93 deg; joints [-7.73, -0.474, 33.474, 96.756, -100.267, 113.608, -1175.929]
  Set speed (1000.0 mm/s)
  MoveL 577 to (-55.37, 234.2, 0) mm, rotated rx 0 ry -90 rz 85.93 deg; joints [-7.73, -0.474, 33.474, 96.756, -100.267, 113.608, -1175.929]
  Set speed (1000.0 mm/s)
  MoveL 578 to (58.93, 255.88, 290) mm, rotated rx 0 ry -90 rz -114.31 deg; joints [0.773, 4.57, 21.856, 99.582, -108.518, 97.992, -1345.694]
  MoveL 579 to (58.93, 255.88, 290) mm, rotated rx 0 ry -90 rz -114.31 deg; joints [0.773, 4.57, 21.856, 99.582, -108.518, 97.992, -1345.694]
  Set speed (60.0 mm/s)
  MoveL 580 to (37.11, 300.24, 290) mm, rotated rx 0 ry -90 rz -66.45 deg; joints [0.74, 5.545, 19.811, 99.211, -108.664, 96.873, -1393.547]
  Set speed (1000.0 mm/s)
  MoveL 581 to (37.11, 300.24, 290) mm, rotated rx 0 ry -90 rz -66.45 deg; joints [0.74, 5.545, 19.811, 99.211, -108.664, 96.873, -1393.547]
  Set speed (1000.0 mm/s)
  MoveL 582 to (-55.37, 234.2, 0) mm, rotated rx 0 ry -90 rz 85.93 deg; joints [-7.73, -0.474, 33.474, 96.756, -100.267, 113.608, -1535.929]
  MoveL 583 to (-55.37, 234.2, 0) mm, rotated rx 0 ry -90 rz 85.93 deg; joints [-7.73, -0.474, 33.474, 96.756, -100.267, 113.608, -1535.929]
  Set speed (60.0 mm/s)
  MoveL 584 to (-20.49, 199.16, 0) mm, rotated rx 0 ry -90 rz 138.05 deg; joints [-7.713, -0.85, 34.304, 96.846, -100.227, 114.067, -1588.047]
  Set speed (1000.0 mm/s)
  MoveL 585 to (-20.49, 199.16, 0) mm, rotated rx 0 ry -90 rz 138.05 deg; joints [-7.713, -0.85, 34.304, 96.846, -100.227, 114.067, -1588.047]
  Set speed (1000.0 mm/s)
  MoveL 586 to (-55.37, 234.2, 0) mm, rotated rx 0 ry -90 rz 85.93 deg; joints [-7.73, -0.474, 33.474, 96.756, -100.267, 113.608, -1535.929]
  MoveL 587 to (-55.37, 234.2, 0) mm, rotated rx 0 ry -90 rz 85.93 deg; joints [-7.73, -0.474, 33.474, 96.756, -100.267, 113.608, -1535.929]
  Set speed (60.0 mm/s)
  MoveL 588 to (-53.73, 230.19, 10) mm, rotated rx 0 ry -90 rz 90.24 deg; joints [-7.443, -0.178, 32.854, 96.857, -100.544, 113.31, -1540.24]
  MoveL 589 to (-51.6, 225.93, 20) mm, rotated rx 0 ry -90 rz 95 deg; joints [-7.158, 0.132, 32.206, 96.953, -100.824, 112.997, -1545.005]
  MoveL 590 to (-48.92, 221.54, 30) mm, rotated rx 0 ry -90 rz 100.19 deg; joints [-6.872, 0.458, 31.525, 97.042, -101.107, 112.669, -1550.192]
  MoveL 591 to (-45.64, 217.12, 40) mm, rotated rx 0 ry -90 rz 105.77 deg; joints [-6.587, 0.803, 30.805, 97.124, -101.394, 112.32, -1555.772]
  MoveL 592 to (-41.73, 212.8, 50) mm, rotated rx 0 ry -90 rz 111.71 deg; joints [-6.303, 1.171, 30.04, 97.198, -101.684, 111.948, -1561.712]
  MoveL 593 to (-37.21, 208.71, 60) mm, rotated rx 0 ry -90 rz 117.98 deg; joints [-6.019, 1.565, 29.218, 97.261, -101.979, 111.546, -1567.979]
  MoveL 594 to (-32.08, 204.97, 70) mm, rotated rx 0 ry -90 rz 124.54 deg; joints [-5.737, 1.992, 28.33, 97.314, -102.279, 111.11, -1574.536]
  MoveL 595 to (-26.38, 201.72, 80) mm, rotated rx 0 ry -90 rz 131.35 deg; joints [-5.455, 2.459, 27.36, 97.352, -102.585, 110.63, -1581.346]
  MoveL 596 to (-20.21, 199.05, 90) mm, rotated rx 0 ry -90 rz 138.37 deg; joints [-5.174, 2.974, 26.29, 97.373, -102.899, 110.098, -1588.366]
  MoveL 597 to (-13.63, 197.08, 100) mm, rotated rx 0 ry -90 rz 145.55 deg; joints [-4.894, 3.55, 25.095, 97.373, -103.221, 109.501, -1595.555]
  MoveL 598 to (-6.77, 195.87, 110) mm, rotated rx 0 ry -90 rz 152.87 deg; joints [-4.615, 4.205, 23.739, 97.347, -103.554, 108.818, -1602.866]
  MoveL 599 to (0.24, 195.48, 120) mm, rotated rx 0 ry -90 rz 160.25 deg; joints [-4.338, 4.966, 22.167, 97.287, -103.902, 108.022, -1610.252]
  MoveL 600 to (7.28, 195.93, 130) mm, rotated rx 0 ry -90 rz 167.67 deg; joints [-4.062, 5.883, 20.277, 97.176, -104.269, 107.059, -1617.666]
  MoveL 601 to (14.2, 197.22, 140) mm, rotated rx 0 ry -90 rz 175.06 deg; joints [-3.787, 7.067, 17.844, 96.983, -104.669, 105.812, -1625.059]
  MoveL 602 to (20.88, 199.3, 150) mm, rotated rx 0 ry -90 rz -177.62 deg; joints [-3.513, 8.962, 13.974, 96.579, -105.151, 103.813, -1632.384]
  MoveL 603 to (26.91, 204.04, 159.43) mm, rotated rx 0 ry -90 rz -170.41 deg; joints [-3.241, 10.894, 10.028, 96.138, -105.625, 101.765, -1639.594]
  MoveL 604 to (31.73, 210.33, 168.53) mm, rotated rx 0 ry -90 rz -163.36 deg; joints [-2.97, 10.872, 10.028, 96.236, -105.879, 101.771, -1646.645]
  MoveL 605 to (38.31, 209.62, 180) mm, rotated rx 0 ry -90 rz -166.51 deg; joints [-2.204, -2.855, 37.416, 100.32, -104.578, 105.885, -1653.494]
  MoveL 606 to (42.97, 214.08, 190) mm, rotated rx 0 ry -90 rz -159.9 deg; joints [-1.929, -2.395, 36.438, 100.352, -104.894, 105.4, -1660.103]
  MoveL 607 to (46.98, 218.83, 200) mm, rotated rx 0 ry -90 rz -153.57 deg; joints [-1.655, -1.908, 35.404, 100.37, -105.217, 104.884, -1666.434]
  MoveL 608 to (50.33, 223.75, 210) mm, rotated rx 0 ry -90 rz -147.55 deg; joints [-1.382, -1.392, 34.309, 100.375, -105.546, 104.337, -1672.453]
  MoveL 609 to (53.04, 228.71, 220) mm, rotated rx 0 ry -90 rz -141.87 deg; joints [-1.11, -0.842, 33.147, 100.363, -105.881, 103.754, -1678.126]
  MoveL 610 to (55.14, 233.59, 230) mm, rotated rx 0 ry -90 rz -136.58 deg; joints [-0.838, -0.257, 31.912, 100.335, -106.224, 103.133, -1683.424]
  MoveL 611 to (56.69, 238.28, 240) mm, rotated rx 0 ry -90 rz -131.68 deg; joints [-0.568, 0.37, 30.593, 100.287, -106.575, 102.466, -1688.316]
  MoveL 612 to (57.77, 242.68, 250) mm, rotated rx 0 ry -90 rz -127.23 deg; joints [-0.299, 1.047, 29.176, 100.217, -106.935, 101.748, -1692.774]
  MoveL 613 to (58.44, 246.7, 260) mm, rotated rx 0 ry -90 rz -123.23 deg; joints [-0.03, 1.782, 27.639, 100.121, -107.307, 100.965, -1696.77]
  MoveL 614 to (58.8, 250.28, 270) mm, rotated rx 0 ry -90 rz -119.73 deg; joints [0.238, 2.594, 25.949, 99.991, -107.691, 100.101, -1700.274]
  MoveL 615 to (58.94, 253.36, 280) mm, rotated rx 0 ry -90 rz -116.74 deg; joints [0.506, 3.507, 24.053, 99.817, -108.092, 99.127, -1703.258]
  MoveL 616 to (58.93, 255.88, 290) mm, rotated rx 0 ry -90 rz -114.31 deg; joints [0.773, 4.57, 21.856, 99.582, -108.518, 97.992, -1705.694]
  Set speed (1000.0 mm/s)
  MoveL 617 to (58.93, 255.88, 290) mm, rotated rx 0 ry -90 rz -114.31 deg; joints [0.773, 4.57, 21.856, 99.582, -108.518, 97.992, -1705.694]
  Set speed (1000.0 mm/s)
  MoveL 618 to (37.11, 300.24, 290) mm, rotated rx 147.65 ry -80.41 rz 116.63 deg; joints [2.261, -4.393, 33.897, 108.752, -102.77, 101.131, -1726.629]
  MoveL 619 to (37.11, 300.24, 290) mm, rotated rx 147.65 ry -80.41 rz 116.63 deg; joints [2.261, -4.393, 33.897, 108.752, -102.77, 101.131, -1726.629]
  Set speed (60.0 mm/s)
  MoveL 620 to (38.82, 298.59, 279.91) mm, rotated rx 155.16 ry -78.45 rz 113.61 deg; joints [1.887, 7.258, 10.028, 107.301, -105.03, 96.941, -1723.609]
  MoveL 621 to (41.29, 296.51, 270) mm, rotated rx 152.18 ry -76.69 rz 110.04 deg; joints [1.97, 15.849, -8.328, 106.26, -107.128, 84.714, -1720.035]
  MoveL 622 to (43.78, 293.91, 260) mm, rotated rx 148.78 ry -75.12 rz 105.96 deg; joints [2.02, 19.511, -16.765, 106.359, -107.972, 76.979, -1715.959]
  MoveL 623 to (46.4, 290.79, 250) mm, rotated rx 154.97 ry -73.74 rz 101.43 deg; joints [1.658, 14.033, -5.88, 109.189, -105.479, 88.821, -1711.425]
  MoveL 624 to (49.06, 287.12, 240) mm, rotated rx 150.79 ry -72.53 rz 96.48 deg; joints [1.686, 18.85, -16.499, 108.777, -106.956, 79.271, -1706.478]
  MoveL 625 to (51.62, 282.9, 230) mm, rotated rx 156.28 ry -71.47 rz 91.16 deg; joints [1.323, 14.146, -7.137, 110.982, -104.655, 89.468, -1701.161]
  MoveL 626 to (48.89, 280.03, 217.93) mm, rotated rx 161.47 ry -70.56 rz 85.52 deg; joints [0.945, 5.511, 10.028, 113.488, -100.657, 102.788, -1695.515]
  MoveL 627 to (56, 272.86, 210) mm, rotated rx 156.39 ry -69.77 rz 79.58 deg; joints [0.967, 15.606, -10.903, 111.979, -104.527, 87.633, -1689.582]
  MoveL 628 to (57.57, 267.12, 200) mm, rotated rx 161.07 ry -69.11 rz 73.4 deg; joints [0.591, 9.937, 0.392, 113.73, -101.727, 97.624, -1683.4]
  MoveL 629 to (58.59, 260.98, 190) mm, rotated rx 155.53 ry -68.55 rz 67.01 deg; joints [0.587, 17.669, -15.692, 112.444, -104.789, 84.311, -1677.009]
  MoveL 630 to (58.95, 254.55, 180) mm, rotated rx 159.8 ry -68.1 rz 60.45 deg; joints [0.214, 14.131, -8.568, 113.635, -102.884, 91.935, -1670.447]
  MoveL 631 to (58.59, 247.92, 170) mm, rotated rx 163.91 ry -67.74 rz 53.75 deg; joints [-0.173, 8.122, 3.48, 114.987, -99.895, 101.562, -1663.752]
  MoveL 632 to (57.45, 241.22, 160) mm, rotated rx 157.88 ry -67.47 rz 46.96 deg; joints [-0.19, 17.379, -15.441, 113.389, -103.741, 86.572, -1656.959]
  MoveL 633 to (55.51, 234.59, 150) mm, rotated rx 161.73 ry -67.28 rz 40.11 deg; joints [-0.575, 14.195, -8.953, 114.198, -101.992, 93.411, -1650.107]
  MoveL 634 to (52.77, 228.15, 140) mm, rotated rx 165.5 ry -67.18 rz 33.23 deg; joints [-0.974, 9.181, 1.181, 115.09, -99.454, 101.763, -1643.231]
  MoveL 635 to (49.26, 222.05, 130) mm, rotated rx 159.2 ry -67.16 rz 26.37 deg; joints [-1.015, 17.892, -16.441, 113.482, -103.081, 87.166, -1636.367]
  MoveL 636 to (45.04, 216.4, 120) mm, rotated rx 162.85 ry -67.22 rz 19.55 deg; joints [-1.416, 15.009, -10.46, 113.987, -101.486, 93.542, -1629.55]
  MoveL 637 to (40.19, 211.31, 110) mm, rotated rx 166.47 ry -67.36 rz 12.82 deg; joints [-1.832, 10.768, -1.782, 114.52, -99.339, 101.084, -1622.816]
  MoveL 638 to (34.83, 206.87, 100) mm, rotated rx 160.09 ry -67.58 rz 6.2 deg; joints [-1.905, 18.644, -17.537, 112.9, -102.525, 87.287, -1616.2]
  MoveL 639 to (29.06, 203.14, 90) mm, rotated rx 127.25 ry -67.89 rz -0.26 deg; joints [-1.835, 32.782, -50.692, 107.443, -109.252, 35.829, -1609.736]
  MoveL 640 to (23.03, 200.17, 80) mm, rotated rx 121.86 ry -68.29 rz -6.54 deg; joints [-2.237, 33.899, -54.267, 106.282, -109.582, 27.688, -1603.458]
  MoveL 641 to (16.86, 197.94, 70) mm, rotated rx 116.74 ry -68.79 rz -12.6 deg; joints [-2.677, 34.682, -57.245, 105.121, -109.735, 20.022, -1597.4]
  MoveL 642 to (10.69, 196.46, 60) mm, rotated rx 121.89 ry -69.39 rz -18.41 deg; joints [-2.902, 34.493, -54.757, 105.325, -108.869, 27.261, -1591.595]
  MoveL 643 to (4.64, 195.67, 50) mm, rotated rx 127.36 ry -70.11 rz -23.92 deg; joints [-3.178, 33.994, -51.69, 105.459, -107.892, 35.026, -1586.075]
  MoveL 644 to (-1.18, 195.49, 40) mm, rotated rx 123.16 ry -70.95 rz -29.13 deg; joints [-3.58, 34.988, -54.422, 104.129, -107.918, 28.683, -1580.872]
  MoveL 645 to (-6.67, 195.86, 30) mm, rotated rx 129.31 ry -71.93 rz -33.98 deg; joints [-3.897, 34.326, -50.761, 104.092, -106.84, 37.498, -1576.017]
